LIN {X 0,Y 291.211,Z 555.04,A -85,B 0,C 180,E1 -17035.414,E2 -17035.414} C_VEL
LIN {X 0,Y 288.825,Z 546.256,A -85,B 0,C 180,E1 -17037.077,E2 -17037.077} C_VEL
LIN {X 0,Y 287.526,Z 542.188,A -85,B 0,C 180,E1 -17037.895,E2 -17037.895} C_VEL
LIN {X 0,Y 286.228,Z 538.806,A -85,B 0,C 180,E1 -17038.607,E2 -17038.607} C_VEL
LIN {X 0,Y 286.024,Z 537.383,A -85,B 0,C 180,E1 -17038.83,E2 -17038.83} C_VEL
LIN {X 0,Y 287.136,Z 533.298,A -85,B 0,C 180,E1 -17042.581,E2 -17042.581} C_VEL
LIN {X 0,Y 287.484,Z 531.734,A -85,B 0,C 180,E1 -17044.214,E2 -17044.214} C_VEL
LIN {X 0,Y 287.652,Z 529.981,A -85,B 0,C 180,E1 -17046.268,E2 -17046.268} C_VEL
LIN {X 0,Y 287.432,Z 527.724,A -85,B 0,C 180,E1 -17049.475,E2 -17049.475} C_VEL
LIN {X 0,Y 287.136,Z 525.711,A -85,B 0,C 180,E1 -17053.263,E2 -17053.263} C_VEL
LIN {X 0,Y 286.89,Z 524.296,A -85,B 0,C 180,E1 -17057.301,E2 -17057.301} C_VEL
LIN {X 0,Y 286.762,Z 523.703,A -85,B 0,C 180,E1 -17060.416,E2 -17060.416} C_VEL
LIN {X 0,Y 286.633,Z 523.532,A -85,B 0,C 180,E1 -17064.012,E2 -17064.012} C_VEL
LIN {X 0,Y 286.375,Z 523.878,A -85,B 0,C 180,E1 -17067.323,E2 -17067.323} C_VEL
LIN {X 0,Y 285.849,Z 524.654,A -85,B 0,C 180,E1 -17070.546,E2 -17070.546} C_VEL
LIN {X 0,Y 285.752,Z 524.986,A -85,B 0,C 180,E1 -17071.256,E2 -17071.256} C_VEL
LIN {X 0,Y 286.798,Z 527.778,A -85,B 0,C 180,E1 -17071.908,E2 -17071.908} C_VEL
LIN {X 0,Y 288.43,Z 530.445,A -85,B 0,C 180,E1 -17072.756,E2 -17072.756} C_VEL
LIN {X 0,Y 291.728,Z 537.483,A -85,B 0,C 180,E1 -17074.575,E2 -17074.575} C_VEL
LIN {X 0,Y 294.518,Z 545.112,A -85,B 0,C 180,E1 -17076.37,E2 -17076.37} C_VEL
LIN {X 0,Y 296.554,Z 553.072,A -85,B 0,C 180,E1 -17078.154,E2 -17078.154} C_VEL
LIN {X 0,Y 297.27,Z 559.717,A -85,B 0,C 180,E1 -17079.591,E2 -17079.591} C_VEL
LIN {X 0,Y 294.87,Z 568.726,A -85,B 0,C 180,E1 -17081.231,E2 -17081.231} C_VEL
LIN {X 0,Y 292.538,Z 575.978,A -85,B 0,C 180,E1 -17082.885,E2 -17082.885} C_VEL
LIN {X 0,Y 290.461,Z 581.891,A -85,B 0,C 180,E1 -17084.564,E2 -17084.564} C_VEL
LIN {X 0,Y 288.308,Z 587.581,A -85,B 0,C 180,E1 -17086.61,E2 -17086.61} C_VEL
LIN {X 0,Y 286.53,Z 591.939,A -85,B 0,C 180,E1 -17088.684,E2 -17088.684} C_VEL
LIN {X 0,Y 285.572,Z 594.044,A -85,B 0,C 180,E1 -17090.08,E2 -17090.08} C_VEL
LIN {X 0,Y 284.557,Z 595.665,A -85,B 0,C 180,E1 -17091.478,E2 -17091.478} C_VEL
LIN {X 0,Y 283.966,Z 596.785,A -85,B 0,C 180,E1 -17092.892,E2 -17092.892} C_VEL
LIN {X 0,Y 283.615,Z 597.465,A -85,B 0,C 180,E1 -17094.312,E2 -17094.312} C_VEL
LIN {X 0,Y 283.193,Z 597.618,A -85,B 0,C 180,E1 -17095.73,E2 -17095.73} C_VEL
LIN {X 0,Y 282.842,Z 597.22,A -85,B 0,C 180,E1 -17097.152,E2 -17097.152} C_VEL
LIN {X 0,Y 282.589,Z 596.363,A -85,B 0,C 180,E1 -17098.575,E2 -17098.575} C_VEL
LIN {X 0,Y 282.487,Z 595.035,A -85,B 0,C 180,E1 -17100,E2 -17100} C_VEL
LIN {X 0,Y 282.504,Z 591.986,A -85,B 0,C 180,E1 -17102.139,E2 -17102.139} C_VEL
LIN {X 0,Y 282.688,Z 587.669,A -85,B 0,C 180,E1 -17104.277,E2 -17104.277} C_VEL
LIN {X 0,Y 282.863,Z 582.104,A -85,B 0,C 180,E1 -17106.359,E2 -17106.359} C_VEL
LIN {X 0,Y 283.372,Z 575.719,A -85,B 0,C 180,E1 -17108.199,E2 -17108.199} C_VEL
LIN {X 0,Y 283.694,Z 569.729,A -85,B 0,C 180,E1 -17109.626,E2 -17109.626} C_VEL
LIN {X 0,Y 284.187,Z 562.583,A -85,B 0,C 180,E1 -17111.05,E2 -17111.05} C_VEL
LIN {X 0,Y 284.761,Z 555.153,A -85,B 0,C 180,E1 -17112.291,E2 -17112.291} C_VEL
LIN {X 0,Y 285.394,Z 546.206,A -85,B 0,C 180,E1 -17113.529,E2 -17113.529} C_VEL
LIN {X 0,Y 285.721,Z 538.903,A -85,B 0,C 180,E1 -17114.364,E2 -17114.364} C_VEL
LIN {X 0,Y 283.996,Z 527.158,A -85,B 0,C 180,E1 -17115.475,E2 -17115.475} C_VEL
LIN {X 0,Y 282.778,Z 517.151,A -85,B 0,C 180,E1 -17116.19,E2 -17116.19} C_VEL
LIN {X 0,Y 282.826,Z 513.933,A -85,B 0,C 180,E1 -17119.217,E2 -17119.217} C_VEL
LIN {X 0,Y 282.999,Z 510.701,A -85,B 0,C 180,E1 -17122.399,E2 -17122.399} C_VEL
LIN {X 0,Y 284.521,Z 515.556,A -85,B 0,C 180,E1 -17125.612,E2 -17125.612} C_VEL
LIN {X 0,Y 284.962,Z 519.302,A -85,B 0,C 180,E1 -17127.943,E2 -17127.943} C_VEL
LIN {X 0,Y 284.495,Z 526.168,A -85,B 0,C 180,E1 -17132.035,E2 -17132.035} C_VEL
LIN {X 0,Y 284.203,Z 530.487,A -85,B 0,C 180,E1 -17134.61,E2 -17134.61} C_VEL
LIN {X 0,Y 287.389,Z 542.62,A -85,B 0,C 180,E1 -17135.629,E2 -17135.629} C_VEL
LIN {X 0,Y 289.327,Z 553.453,A -85,B 0,C 180,E1 -17136.716,E2 -17136.716} C_VEL
LIN {X 0,Y 290.316,Z 563.05,A -85,B 0,C 180,E1 -17137.9,E2 -17137.9} C_VEL
LIN {X 0,Y 289.367,Z 571.259,A -85,B 0,C 180,E1 -17138.994,E2 -17138.994} C_VEL
LIN {X 0,Y 288.311,Z 578.189,A -85,B 0,C 180,E1 -17140.109,E2 -17140.109} C_VEL
LIN {X 0,Y 287.18,Z 584.655,A -85,B 0,C 180,E1 -17141.358,E2 -17141.358} C_VEL
LIN {X 0,Y 286.044,Z 590.927,A -85,B 0,C 180,E1 -17142.831,E2 -17142.831} C_VEL
LIN {X 0,Y 284.861,Z 597.457,A -85,B 0,C 180,E1 -17144.744,E2 -17144.744} C_VEL
LIN {X 0,Y 284.018,Z 602.375,A -85,B 0,C 180,E1 -17146.632,E2 -17146.632} C_VEL
LIN {X 0,Y 283.441,Z 605.324,A -85,B 0,C 180,E1 -17148.061,E2 -17148.061} C_VEL
LIN {X 0,Y 282.763,Z 608.747,A -85,B 0,C 180,E1 -17150.399,E2 -17150.399} C_VEL
LIN {X 0,Y 282.524,Z 609.981,A -85,B 0,C 180,E1 -17151.545,E2 -17151.545} C_VEL
LIN {X 0,Y 282.249,Z 611.122,A -85,B 0,C 180,E1 -17153.301,E2 -17153.301} C_VEL
LIN {X 0,Y 282.073,Z 611.479,A -85,B 0,C 180,E1 -17155.307,E2 -17155.307} C_VEL
LIN {X 0,Y 282.055,Z 611.13,A -85,B 0,C 180,E1 -17156.757,E2 -17156.757} C_VEL
LIN {X 0,Y 282.192,Z 610.034,A -85,B 0,C 180,E1 -17158.465,E2 -17158.465} C_VEL
LIN {X 0,Y 282.508,Z 607.716,A -85,B 0,C 180,E1 -17160.54,E2 -17160.54} C_VEL
LIN {X 0,Y 282.899,Z 604.085,A -85,B 0,C 180,E1 -17162.639,E2 -17162.639} C_VEL
LIN {X 0,Y 283.415,Z 599.288,A -85,B 0,C 180,E1 -17164.674,E2 -17164.674} C_VEL
LIN {X 0,Y 284.035,Z 594.448,A -85,B 0,C 180,E1 -17166.278,E2 -17166.278} C_VEL
LIN {X 0,Y 284.958,Z 586.826,A -85,B 0,C 180,E1 -17168.287,E2 -17168.287} C_VEL
LIN {X 0,Y 285.914,Z 578.988,A -85,B 0,C 180,E1 -17169.87,E2 -17169.87} C_VEL
LIN {X 0,Y 286.727,Z 571.873,A -85,B 0,C 180,E1 -17171.048,E2 -17171.048} C_VEL
LIN {X 0,Y 287.571,Z 563.23,A -85,B 0,C 180,E1 -17172.212,E2 -17172.212} C_VEL
LIN {X 0,Y 287.615,Z 558.748,A -85,B 0,C 180,E1 -17172.747,E2 -17172.747} C_VEL
LIN {X 0,Y 286.355,Z 548.562,A -85,B 0,C 180,E1 -17173.788,E2 -17173.788} C_VEL
LIN {X 0,Y 284.926,Z 539.502,A -85,B 0,C 180,E1 -17174.524,E2 -17174.524} C_VEL
LIN {X 0,Y 283.266,Z 530.265,A -85,B 0,C 180,E1 -17175.15,E2 -17175.15} C_VEL
LIN {X 0,Y 283.623,Z 523.602,A -85,B 0,C 180,E1 -17179.289,E2 -17179.289} C_VEL
LIN {X 0,Y 283.963,Z 516.651,A -85,B 0,C 180,E1 -17183.605,E2 -17183.605} C_VEL
LIN {X 0,Y 284.284,Z 510.406,A -85,B 0,C 180,E1 -17187.52,E2 -17187.52} C_VEL
LIN {X 0,Y 284.346,Z 509.879,A -85,B 0,C 180,E1 -17187.875,E2 -17187.875} C_VEL
LIN {X 0,Y 284.838,Z 509.818,A -85,B 0,C 180,E1 -17189.999,E2 -17189.999} C_VEL
LIN {X 0,Y 284.746,Z 509.827,A -85,B 0,C 180,E1 -17192.829,E2 -17192.829} C_VEL
LIN {X 0,Y 284.7,Z 509.832,A -85,B 0,C 180,E1 -17197.089,E2 -17197.089} C_VEL
LIN {X 0,Y 284.568,Z 509.85,A -85,B 0,C 180,E1 -17199.955,E2 -17199.955} C_VEL
LIN {X 0,Y 284.482,Z 509.863,A -85,B 0,C 180,E1 -17204.302,E2 -17204.302} C_VEL
LIN {X 0,Y 284.426,Z 509.865,A -85,B 0,C 180,E1 -17207.248,E2 -17207.248} C_VEL
LIN {X 0,Y 284.379,Z 509.876,A -85,B 0,C 180,E1 -17210.241,E2 -17210.241} C_VEL
LIN {X 0,Y 284.369,Z 509.874,A -85,B 0,C 180,E1 -17213.875,E2 -17213.875} C_VEL
LIN {X 0,Y 284.364,Z 509.877,A -85,B 0,C 180,E1 -17218.006,E2 -17218.006} C_VEL
LIN {X 0,Y 284.296,Z 509.882,A -85,B 0,C 180,E1 -17221.273,E2 -17221.273} C_VEL
LIN {X 0,Y 284.36,Z 509.873,A -85,B 0,C 180,E1 -17225.353,E2 -17225.353} C_VEL
LIN {X 0,Y 284.322,Z 509.883,A -85,B 0,C 180,E1 -17228.166,E2 -17228.166} C_VEL
LIN {X 0,Y 284.298,Z 509.884,A -85,B 0,C 180,E1 -17232.131,E2 -17232.131} C_VEL
LIN {X 0,Y 284.317,Z 509.883,A -85,B 0,C 180,E1 -17236.201,E2 -17236.201} C_VEL
LIN {X 0,Y 284.349,Z 509.879,A -85,B 0,C 180,E1 -17240.013,E2 -17240.013} C_VEL
LIN {X 0,Y 284.353,Z 509.874,A -85,B 0,C 180,E1 -17243.617,E2 -17243.617} C_VEL
LIN {X 0,Y 284.305,Z 509.88,A -85,B 0,C 180,E1 -17247.189,E2 -17247.189} C_VEL
LIN {X 0,Y 284.356,Z 509.876,A -85,B 0,C 180,E1 -17250.376,E2 -17250.376} C_VEL
LIN {X 0,Y 284.376,Z 509.873,A -85,B 0,C 180,E1 -17253.586,E2 -17253.586} C_VEL
LIN {X 0,Y 284.364,Z 509.873,A -85,B 0,C 180,E1 -17256.707,E2 -17256.707} C_VEL
LIN {X 0,Y 284.401,Z 509.868,A -85,B 0,C 180,E1 -17261.261,E2 -17261.261} C_VEL
LIN {X 0,Y 284.49,Z 509.858,A -85,B 0,C 180,E1 -17264.459,E2 -17264.459} C_VEL
LIN {X 0,Y 284.487,Z 509.857,A -85,B 0,C 180,E1 -17268.601,E2 -17268.601} C_VEL
LIN {X 0,Y 284.657,Z 509.839,A -85,B 0,C 180,E1 -17271.481,E2 -17271.481} C_VEL
LIN {X 0,Y 284.6,Z 509.845,A -85,B 0,C 180,E1 -17274.331,E2 -17274.331} C_VEL
LIN {X 0,Y 284.855,Z 509.809,A -85,B 0,C 180,E1 -17278.586,E2 -17278.586} C_VEL
LIN {X 0,Y 284.854,Z 509.813,A -85,B 0,C 180,E1 -17281.414,E2 -17281.414} C_VEL
LIN {X 0,Y 284.522,Z 509.854,A -85,B 0,C 180,E1 -17284.135,E2 -17284.135} C_VEL
LIN {X 0,Y 283.792,Z 509.952,A -85,B 0,C 180,E1 -17285.317,E2 -17285.317} C_VEL
LIN {X 0,Y 280.998,Z 510.303,A -85,B 0,C 180,E1 -17287.245,E2 -17287.245} C_VEL
LIN {X 0,Y 277.838,Z 510.69,A -85,B 0,C 180,E1 -17289.614,E2 -17289.614} C_VEL
LIN {X 0,Y 277.482,Z 510.731,A -85,B 0,C 180,E1 -17290.431,E2 -17290.431} C_VEL
LIN {X 0,Y 277.432,Z 510.737,A -85,B 0,C 180,E1 -17294.674,E2 -17294.674} C_VEL
LIN {X 0,Y 277.342,Z 510.75,A -85,B 0,C 180,E1 -17299.234,E2 -17299.234} C_VEL
LIN {X 0,Y 277.326,Z 510.753,A -85,B 0,C 180,E1 -17303.921,E2 -17303.921} C_VEL
LIN {X 0,Y 277.323,Z 510.755,A -85,B 0,C 180,E1 -17307.506,E2 -17307.506} C_VEL
LIN {X 0,Y 277.269,Z 510.758,A -85,B 0,C 180,E1 -17310.482,E2 -17310.482} C_VEL
LIN {X 0,Y 277.252,Z 510.761,A -85,B 0,C 180,E1 -17313.895,E2 -17313.895} C_VEL
LIN {X 0,Y 277.279,Z 510.76,A -85,B 0,C 180,E1 -17317.467,E2 -17317.467} C_VEL
LIN {X 0,Y 277.224,Z 510.766,A -85,B 0,C 180,E1 -17321.234,E2 -17321.234} C_VEL
LIN {X 0,Y 277.231,Z 510.765,A -85,B 0,C 180,E1 -17325.22,E2 -17325.22} C_VEL
LIN {X 0,Y 277.285,Z 510.76,A -85,B 0,C 180,E1 -17329.497,E2 -17329.497} C_VEL
LIN {X 0,Y 277.513,Z 510.799,A -85,B 0,C 180,E1 -17332.163,E2 -17332.163} C_VEL
LIN {X 0,Y 278.528,Z 516.826,A -85,B 0,C 180,E1 -17336.375,E2 -17336.375} C_VEL
LIN {X 0,Y 278.767,Z 519.283,A -85,B 0,C 180,E1 -17338.034,E2 -17338.034} C_VEL
LIN {X 0,Y 277.963,Z 524.259,A -85,B 0,C 180,E1 -17341.29,E2 -17341.29} C_VEL
LIN {X 0,Y 276.905,Z 531.592,A -85,B 0,C 180,E1 -17346.042,E2 -17346.042} C_VEL
LIN {X 0,Y 276.175,Z 538.547,A -85,B 0,C 180,E1 -17350.515,E2 -17350.515} C_VEL
LIN {X 0,Y 277.843,Z 552.725,A -85,B 0,C 180,E1 -17351.234,E2 -17351.234} C_VEL
LIN {X 0,Y 278.722,Z 562.025,A -85,B 0,C 180,E1 -17351.914,E2 -17351.914} C_VEL
LIN {X 0,Y 279.238,Z 570.27,A -85,B 0,C 180,E1 -17352.681,E2 -17352.681} C_VEL
LIN {X 0,Y 279.551,Z 579.34,A -85,B 0,C 180,E1 -17353.732,E2 -17353.732} C_VEL
LIN {X 0,Y 279.2,Z 586.143,A -85,B 0,C 180,E1 -17354.675,E2 -17354.675} C_VEL
LIN {X 0,Y 278.266,Z 593.763,A -85,B 0,C 180,E1 -17355.932,E2 -17355.932} C_VEL
LIN {X 0,Y 277.355,Z 601.745,A -85,B 0,C 180,E1 -17357.563,E2 -17357.563} C_VEL
LIN {X 0,Y 276.494,Z 608.666,A -85,B 0,C 180,E1 -17359.381,E2 -17359.381} C_VEL
LIN {X 0,Y 275.949,Z 614.155,A -85,B 0,C 180,E1 -17361.211,E2 -17361.211} C_VEL
LIN {X 0,Y 275.503,Z 619.232,A -85,B 0,C 180,E1 -17363.409,E2 -17363.409} C_VEL
LIN {X 0,Y 275.325,Z 622.886,A -85,B 0,C 180,E1 -17365.609,E2 -17365.609} C_VEL
LIN {X 0,Y 275.323,Z 624.523,A -85,B 0,C 180,E1 -17367.074,E2 -17367.074} C_VEL
LIN {X 0,Y 275.3,Z 625.615,A -85,B 0,C 180,E1 -17368.538,E2 -17368.538} C_VEL
LIN {X 0,Y 275.325,Z 626.211,A -85,B 0,C 180,E1 -17370.001,E2 -17370.001} C_VEL
LIN {X 0,Y 275.297,Z 626.32,A -85,B 0,C 180,E1 -17371.464,E2 -17371.464} C_VEL
LIN {X 0,Y 275.314,Z 625.931,A -85,B 0,C 180,E1 -17372.927,E2 -17372.927} C_VEL
LIN {X 0,Y 275.319,Z 624.951,A -85,B 0,C 180,E1 -17374.393,E2 -17374.393} C_VEL
LIN {X 0,Y 275.524,Z 622.567,A -85,B 0,C 180,E1 -17376.592,E2 -17376.592} C_VEL
LIN {X 0,Y 275.695,Z 621.412,A -85,B 0,C 180,E1 -17377.324,E2 -17377.324} C_VEL
LIN {X 0,Y 276.68,Z 617.967,A -85,B 0,C 180,E1 -17380.243,E2 -17380.243} C_VEL
LIN {X 0,Y 277.921,Z 614.293,A -85,B 0,C 180,E1 -17382.413,E2 -17382.413} C_VEL
LIN {X 0,Y 279.712,Z 609.31,A -85,B 0,C 180,E1 -17384.553,E2 -17384.553} C_VEL
LIN {X 0,Y 281.526,Z 604.159,A -85,B 0,C 180,E1 -17386.311,E2 -17386.311} C_VEL
LIN {X 0,Y 283.064,Z 599.285,A -85,B 0,C 180,E1 -17387.708,E2 -17387.708} C_VEL
LIN {X 0,Y 285.508,Z 591.962,A -85,B 0,C 180,E1 -17389.41,E2 -17389.41} C_VEL
LIN {X 0,Y 287.159,Z 584.573,A -85,B 0,C 180,E1 -17390.942,E2 -17390.942} C_VEL
LIN {X 0,Y 287.682,Z 577.918,A -85,B 0,C 180,E1 -17392.251,E2 -17392.251} C_VEL
LIN {X 0,Y 287.227,Z 567.044,A -85,B 0,C 180,E1 -17394.369,E2 -17394.369} C_VEL
LIN {X 0,Y 285.224,Z 555.475,A -85,B 0,C 180,E1 -17396.633,E2 -17396.633} C_VEL
LIN {X 0,Y 283.08,Z 547.236,A -85,B 0,C 180,E1 -17398.356,E2 -17398.356} C_VEL
LIN {X 0,Y 281.383,Z 541.883,A -85,B 0,C 180,E1 -17399.585,E2 -17399.585} C_VEL
LIN {X 0,Y 279.978,Z 538.608,A -85,B 0,C 180,E1 -17400.431,E2 -17400.431} C_VEL
LIN {X 0,Y 279.641,Z 536.505,A -85,B 0,C 180,E1 -17400.87,E2 -17400.87} C_VEL
LIN {X 0,Y 280.553,Z 533.19,A -85,B 0,C 180,E1 -17404.242,E2 -17404.242} C_VEL
LIN {X 0,Y 280.668,Z 531.012,A -85,B 0,C 180,E1 -17406.94,E2 -17406.94} C_VEL
LIN {X 0,Y 280.419,Z 528.637,A -85,B 0,C 180,E1 -17410.665,E2 -17410.665} C_VEL
LIN {X 0,Y 280.162,Z 526.796,A -85,B 0,C 180,E1 -17414.62,E2 -17414.62} C_VEL
LIN {X 0,Y 279.985,Z 525.939,A -85,B 0,C 180,E1 -17417.333,E2 -17417.333} C_VEL
LIN {X 0,Y 279.822,Z 525.264,A -85,B 0,C 180,E1 -17421.133,E2 -17421.133} C_VEL
LIN {X 0,Y 279.635,Z 525.177,A -85,B 0,C 180,E1 -17424.686,E2 -17424.686} C_VEL
LIN {X 0,Y 279.316,Z 525.596,A -85,B 0,C 180,E1 -17428.103,E2 -17428.103} C_VEL
LIN {X 0,Y 279.229,Z 525.917,A -85,B 0,C 180,E1 -17429.208,E2 -17429.208} C_VEL
LIN {X 0,Y 280.088,Z 528.435,A -85,B 0,C 180,E1 -17429.878,E2 -17429.878} C_VEL
LIN {X 0,Y 281.728,Z 530.717,A -85,B 0,C 180,E1 -17430.824,E2 -17430.824} C_VEL
LIN {X 0,Y 285.489,Z 538.633,A -85,B 0,C 180,E1 -17433.195,E2 -17433.195} C_VEL
LIN {X 0,Y 288.139,Z 545.714,A -85,B 0,C 180,E1 -17435.074,E2 -17435.074} C_VEL
LIN {X 0,Y 290.208,Z 553.385,A -85,B 0,C 180,E1 -17436.964,E2 -17436.964} C_VEL
LIN {X 0,Y 291.107,Z 559.638,A -85,B 0,C 180,E1 -17438.451,E2 -17438.451} C_VEL
LIN {X 0,Y 291.107,Z 562.823,A -85,B 0,C 180,E1 -17439.139,E2 -17439.139} C_VEL
LIN {X 0,Y 288.431,Z 571.16,A -85,B 0,C 180,E1 -17440.795,E2 -17440.795} C_VEL
LIN {X 0,Y 286.006,Z 577.979,A -85,B 0,C 180,E1 -17442.481,E2 -17442.481} C_VEL
LIN {X 0,Y 283.824,Z 583.652,A -85,B 0,C 180,E1 -17444.194,E2 -17444.194} C_VEL
LIN {X 0,Y 281.553,Z 589.068,A -85,B 0,C 180,E1 -17446.283,E2 -17446.283} C_VEL
LIN {X 0,Y 279.655,Z 593.016,A -85,B 0,C 180,E1 -17448.402,E2 -17448.402} C_VEL
LIN {X 0,Y 278.651,Z 595.054,A -85,B 0,C 180,E1 -17449.831,E2 -17449.831} C_VEL
LIN {X 0,Y 277.602,Z 596.516,A -85,B 0,C 180,E1 -17451.263,E2 -17451.263} C_VEL
LIN {X 0,Y 276.958,Z 597.456,A -85,B 0,C 180,E1 -17452.711,E2 -17452.711} C_VEL
LIN {X 0,Y 276.566,Z 597.945,A -85,B 0,C 180,E1 -17454.166,E2 -17454.166} C_VEL
LIN {X 0,Y 276.131,Z 598.009,A -85,B 0,C 180,E1 -17455.621,E2 -17455.621} C_VEL
LIN {X 0,Y 275.768,Z 597.514,A -85,B 0,C 180,E1 -17457.078,E2 -17457.078} C_VEL
LIN {X 0,Y 275.508,Z 596.486,A -85,B 0,C 180,E1 -17458.538,E2 -17458.538} C_VEL
LIN {X 0,Y 275.404,Z 594.989,A -85,B 0,C 180,E1 -17460,E2 -17460} C_VEL
LIN {X 0,Y 275.431,Z 591.762,A -85,B 0,C 180,E1 -17462.194,E2 -17462.194} C_VEL
LIN {X 0,Y 275.609,Z 587.285,A -85,B 0,C 180,E1 -17464.388,E2 -17464.388} C_VEL
LIN {X 0,Y 275.776,Z 582.036,A -85,B 0,C 180,E1 -17466.33,E2 -17466.33} C_VEL
LIN {X 0,Y 276.255,Z 576.21,A -85,B 0,C 180,E1 -17468.043,E2 -17468.043} C_VEL
LIN {X 0,Y 276.545,Z 570.229,A -85,B 0,C 180,E1 -17469.508,E2 -17469.508} C_VEL
LIN {X 0,Y 277.073,Z 563.111,A -85,B 0,C 180,E1 -17470.967,E2 -17470.967} C_VEL
LIN {X 0,Y 277.715,Z 554.54,A -85,B 0,C 180,E1 -17472.422,E2 -17472.422} C_VEL
LIN {X 0,Y 278.479,Z 544.006,A -85,B 0,C 180,E1 -17473.872,E2 -17473.872} C_VEL
LIN {X 0,Y 278.594,Z 539.019,A -85,B 0,C 180,E1 -17474.425,E2 -17474.425} C_VEL
LIN {X 0,Y 276.917,Z 527.605,A -85,B 0,C 180,E1 -17475.534,E2 -17475.534} C_VEL
LIN {X 0,Y 275.698,Z 517.493,A -85,B 0,C 180,E1 -17476.285,E2 -17476.285} C_VEL
LIN {X 0,Y 275.741,Z 514.209,A -85,B 0,C 180,E1 -17479.428,E2 -17479.428} C_VEL
LIN {X 0,Y 275.868,Z 511.733,A -85,B 0,C 180,E1 -17481.924,E2 -17481.924} C_VEL
LIN {X 0,Y 277.571,Z 516.984,A -85,B 0,C 180,E1 -17485.495,E2 -17485.495} C_VEL
LIN {X 0,Y 278.021,Z 520.527,A -85,B 0,C 180,E1 -17487.777,E2 -17487.777} C_VEL
LIN {X 0,Y 277.505,Z 527.693,A -85,B 0,C 180,E1 -17492.13,E2 -17492.13} C_VEL
LIN {X 0,Y 277.289,Z 530.831,A -85,B 0,C 180,E1 -17493.945,E2 -17493.945} C_VEL
LIN {X 0,Y 280.094,Z 540.854,A -85,B 0,C 180,E1 -17494.808,E2 -17494.808} C_VEL
LIN {X 0,Y 281.952,Z 549.804,A -85,B 0,C 180,E1 -17495.712,E2 -17495.712} C_VEL
LIN {X 0,Y 283.431,Z 560.979,A -85,B 0,C 180,E1 -17497.033,E2 -17497.033} C_VEL
LIN {X 0,Y 283.585,Z 565.7,A -85,B 0,C 180,E1 -17497.685,E2 -17497.685} C_VEL
LIN {X 0,Y 282.101,Z 575.692,A -85,B 0,C 180,E1 -17499.136,E2 -17499.136} C_VEL
LIN {X 0,Y 280.706,Z 583.539,A -85,B 0,C 180,E1 -17500.614,E2 -17500.614} C_VEL
LIN {X 0,Y 279.484,Z 589.911,A -85,B 0,C 180,E1 -17502.087,E2 -17502.087} C_VEL
LIN {X 0,Y 278.529,Z 594.928,A -85,B 0,C 180,E1 -17503.494,E2 -17503.494} C_VEL
LIN {X 0,Y 277.593,Z 599.734,A -85,B 0,C 180,E1 -17505.145,E2 -17505.145} C_VEL
LIN {X 0,Y 276.862,Z 603.456,A -85,B 0,C 180,E1 -17506.734,E2 -17506.734} C_VEL
LIN {X 0,Y 276.198,Z 606.799,A -85,B 0,C 180,E1 -17508.578,E2 -17508.578} C_VEL
LIN {X 0,Y 275.685,Z 609.201,A -85,B 0,C 180,E1 -17510.407,E2 -17510.407} C_VEL
LIN {X 0,Y 275.32,Z 610.81,A -85,B 0,C 180,E1 -17512.31,E2 -17512.31} C_VEL
LIN {X 0,Y 275.005,Z 611.686,A -85,B 0,C 180,E1 -17514.864,E2 -17514.864} C_VEL
LIN {X 0,Y 275.012,Z 610.826,A -85,B 0,C 180,E1 -17517.543,E2 -17517.543} C_VEL
LIN {X 0,Y 275.374,Z 608.378,A -85,B 0,C 180,E1 -17520.197,E2 -17520.197} C_VEL
LIN {X 0,Y 275.83,Z 604.317,A -85,B 0,C 180,E1 -17522.7,E2 -17522.7} C_VEL
LIN {X 0,Y 276.214,Z 600.612,A -85,B 0,C 180,E1 -17524.37,E2 -17524.37} C_VEL
LIN {X 0,Y 276.846,Z 595.913,A -85,B 0,C 180,E1 -17526.05,E2 -17526.05} C_VEL
LIN {X 0,Y 277.541,Z 590.292,A -85,B 0,C 180,E1 -17527.676,E2 -17527.676} C_VEL
LIN {X 0,Y 278.312,Z 584.201,A -85,B 0,C 180,E1 -17529.121,E2 -17529.121} C_VEL
LIN {X 0,Y 279.177,Z 577.064,A -85,B 0,C 180,E1 -17530.515,E2 -17530.515} C_VEL
LIN {X 0,Y 280.286,Z 567.591,A -85,B 0,C 180,E1 -17532.003,E2 -17532.003} C_VEL
LIN {X 0,Y 280.754,Z 560.552,A -85,B 0,C 180,E1 -17532.894,E2 -17532.894} C_VEL
LIN {X 0,Y 279.468,Z 549.59,A -85,B 0,C 180,E1 -17534.076,E2 -17534.076} C_VEL
LIN {X 0,Y 277.943,Z 539.973,A -85,B 0,C 180,E1 -17534.892,E2 -17534.892} C_VEL
LIN {X 0,Y 276.226,Z 530.431,A -85,B 0,C 180,E1 -17535.533,E2 -17535.533} C_VEL
LIN {X 0,Y 276.614,Z 523.757,A -85,B 0,C 180,E1 -17539.755,E2 -17539.755} C_VEL
LIN {X 0,Y 276.913,Z 517.912,A -85,B 0,C 180,E1 -17543.441,E2 -17543.441} C_VEL
LIN {X 0,Y 277.195,Z 512.161,A -85,B 0,C 180,E1 -17547.093,E2 -17547.093} C_VEL
LIN {X 0,Y 277.335,Z 510.753,A -85,B 0,C 180,E1 -17548.002,E2 -17548.002} C_VEL
LIN {X 0,Y 277.796,Z 510.695,A -85,B 0,C 180,E1 -17549.999,E2 -17549.999} C_VEL
LIN {X 0,Y 277.702,Z 510.705,A -85,B 0,C 180,E1 -17552.901,E2 -17552.901} C_VEL
LIN {X 0,Y 277.655,Z 510.709,A -85,B 0,C 180,E1 -17557.27,E2 -17557.27} C_VEL
LIN {X 0,Y 277.508,Z 510.732,A -85,B 0,C 180,E1 -17560.21,E2 -17560.21} C_VEL
LIN {X 0,Y 277.435,Z 510.738,A -85,B 0,C 180,E1 -17564.673,E2 -17564.673} C_VEL
LIN {X 0,Y 277.345,Z 510.747,A -85,B 0,C 180,E1 -17569.233,E2 -17569.233} C_VEL
LIN {X 0,Y 277.319,Z 510.754,A -85,B 0,C 180,E1 -17574.17,E2 -17574.17} C_VEL
LIN {X 0,Y 277.335,Z 510.749,A -85,B 0,C 180,E1 -17577.508,E2 -17577.508} C_VEL
LIN {X 0,Y 277.271,Z 510.759,A -85,B 0,C 180,E1 -17580.481,E2 -17580.481} C_VEL
LIN {X 0,Y 277.253,Z 510.761,A -85,B 0,C 180,E1 -17583.894,E2 -17583.894} C_VEL
LIN {X 0,Y 277.28,Z 510.756,A -85,B 0,C 180,E1 -17587.466,E2 -17587.466} C_VEL
LIN {X 0,Y 277.233,Z 510.761,A -85,B 0,C 180,E1 -17591.231,E2 -17591.231} C_VEL
LIN {X 0,Y 277.249,Z 510.759,A -85,B 0,C 180,E1 -17595.215,E2 -17595.215} C_VEL
LIN {X 0,Y 277.293,Z 510.755,A -85,B 0,C 180,E1 -17599.494,E2 -17599.494} C_VEL
LIN {X 0,Y 277.288,Z 510.753,A -85,B 0,C 180,E1 -17602.534,E2 -17602.534} C_VEL
LIN {X 0,Y 277.252,Z 510.763,A -85,B 0,C 180,E1 -17606.105,E2 -17606.105} C_VEL
LIN {X 0,Y 277.259,Z 510.76,A -85,B 0,C 180,E1 -17609.538,E2 -17609.538} C_VEL
LIN {X 0,Y 277.356,Z 510.745,A -85,B 0,C 180,E1 -17612.864,E2 -17612.864} C_VEL
LIN {X 0,Y 277.326,Z 510.754,A -85,B 0,C 180,E1 -17616.079,E2 -17616.079} C_VEL
LIN {X 0,Y 277.342,Z 510.746,A -85,B 0,C 180,E1 -17620.766,E2 -17620.766} C_VEL
LIN {X 0,Y 277.432,Z 510.738,A -85,B 0,C 180,E1 -17625.326,E2 -17625.326} C_VEL
LIN {X 0,Y 277.505,Z 510.731,A -85,B 0,C 180,E1 -17629.789,E2 -17629.789} C_VEL
LIN {X 0,Y 277.651,Z 510.709,A -85,B 0,C 180,E1 -17632.729,E2 -17632.729} C_VEL
LIN {X 0,Y 277.821,Z 510.685,A -85,B 0,C 180,E1 -17638.55,E2 -17638.55} C_VEL
LIN {X 0,Y 277.819,Z 510.689,A -85,B 0,C 180,E1 -17641.449,E2 -17641.449} C_VEL
LIN {X 0,Y 277.651,Z 510.71,A -85,B 0,C 180,E1 -17647.271,E2 -17647.271} C_VEL
LIN {X 0,Y 277.482,Z 510.731,A -85,B 0,C 180,E1 -17650.431,E2 -17650.431} C_VEL
LIN {X 0,Y 276.754,Z 510.826,A -85,B 0,C 180,E1 -17651.641,E2 -17651.641} C_VEL
LIN {X 0,Y 273.911,Z 511.18,A -85,B 0,C 180,E1 -17653.614,E2 -17653.614} C_VEL
LIN {X 0,Y 271.509,Z 511.478,A -85,B 0,C 180,E1 -17655.216,E2 -17655.216} C_VEL
LIN {X 0,Y 270.438,Z 511.608,A -85,B 0,C 180,E1 -17656.457,E2 -17656.457} C_VEL
LIN {X 0,Y 270.327,Z 511.62,A -85,B 0,C 180,E1 -17656.878,E2 -17656.878} C_VEL
LIN {X 0,Y 270.29,Z 511.627,A -85,B 0,C 180,E1 -17660.602,E2 -17660.602} C_VEL
LIN {X 0,Y 270.271,Z 511.629,A -85,B 0,C 180,E1 -17664.586,E2 -17664.586} C_VEL
LIN {X 0,Y 270.267,Z 511.632,A -85,B 0,C 180,E1 -17667.909,E2 -17667.909} C_VEL
LIN {X 0,Y 270.182,Z 511.643,A -85,B 0,C 180,E1 -17671.348,E2 -17671.348} C_VEL
LIN {X 0,Y 270.212,Z 511.637,A -85,B 0,C 180,E1 -17674.904,E2 -17674.904} C_VEL
LIN {X 0,Y 270.219,Z 511.635,A -85,B 0,C 180,E1 -17678.717,E2 -17678.717} C_VEL
LIN {X 0,Y 270.189,Z 511.64,A -85,B 0,C 180,E1 -17682.555,E2 -17682.555} C_VEL
LIN {X 0,Y 270.195,Z 511.639,A -85,B 0,C 180,E1 -17686.744,E2 -17686.744} C_VEL
LIN {X 0,Y 270.426,Z 511.613,A -85,B 0,C 180,E1 -17691.887,E2 -17691.887} C_VEL
LIN {X 0,Y 270.496,Z 511.898,A -85,B 0,C 180,E1 -17692.37,E2 -17692.37} C_VEL
LIN {X 0,Y 271.355,Z 516.902,A -85,B 0,C 180,E1 -17695.974,E2 -17695.974} C_VEL
LIN {X 0,Y 271.684,Z 519.735,A -85,B 0,C 180,E1 -17697.956,E2 -17697.956} C_VEL
LIN {X 0,Y 270.853,Z 524.703,A -85,B 0,C 180,E1 -17701.3,E2 -17701.3} C_VEL
LIN {X 0,Y 269.858,Z 531.321,A -85,B 0,C 180,E1 -17705.716,E2 -17705.716} C_VEL
LIN {X 0,Y 269.118,Z 537.883,A -85,B 0,C 180,E1 -17710.074,E2 -17710.074} C_VEL
LIN {X 0,Y 270.83,Z 552.126,A -85,B 0,C 180,E1 -17710.803,E2 -17710.803} C_VEL
LIN {X 0,Y 271.71,Z 561.831,A -85,B 0,C 180,E1 -17711.528,E2 -17711.528} C_VEL
LIN {X 0,Y 272.284,Z 570.584,A -85,B 0,C 180,E1 -17712.373,E2 -17712.373} C_VEL
LIN {X 0,Y 272.543,Z 578.73,A -85,B 0,C 180,E1 -17713.344,E2 -17713.344} C_VEL
LIN {X 0,Y 272.446,Z 584.136,A -85,B 0,C 180,E1 -17714.094,E2 -17714.094} C_VEL
LIN {X 0,Y 271.515,Z 592.063,A -85,B 0,C 180,E1 -17715.383,E2 -17715.383} C_VEL
LIN {X 0,Y 270.783,Z 597.757,A -85,B 0,C 180,E1 -17716.492,E2 -17716.492} C_VEL
LIN {X 0,Y 270.025,Z 604.102,A -85,B 0,C 180,E1 -17717.983,E2 -17717.983} C_VEL
LIN {X 0,Y 269.356,Z 609.357,A -85,B 0,C 180,E1 -17719.477,E2 -17719.477} C_VEL
LIN {X 0,Y 268.91,Z 613.727,A -85,B 0,C 180,E1 -17720.979,E2 -17720.979} C_VEL
LIN {X 0,Y 268.425,Z 618.852,A -85,B 0,C 180,E1 -17723.234,E2 -17723.234} C_VEL
LIN {X 0,Y 268.236,Z 622.569,A -85,B 0,C 180,E1 -17725.493,E2 -17725.493} C_VEL
LIN {X 0,Y 268.233,Z 624.232,A -85,B 0,C 180,E1 -17726.997,E2 -17726.997} C_VEL
LIN {X 0,Y 268.226,Z 625.365,A -85,B 0,C 180,E1 -17728.499,E2 -17728.499} C_VEL
LIN {X 0,Y 268.247,Z 626,A -85,B 0,C 180,E1 -17730.001,E2 -17730.001} C_VEL
LIN {X 0,Y 268.223,Z 626.148,A -85,B 0,C 180,E1 -17731.502,E2 -17731.502} C_VEL
LIN {X 0,Y 268.225,Z 625.777,A -85,B 0,C 180,E1 -17733.005,E2 -17733.005} C_VEL
LIN {X 0,Y 268.344,Z 623.805,A -85,B 0,C 180,E1 -17735.6,E2 -17735.6} C_VEL
LIN {X 0,Y 270.111,Z 617.084,A -85,B 0,C 180,E1 -17741.254,E2 -17741.254} C_VEL
LIN {X 0,Y 271.567,Z 613.248,A -85,B 0,C 180,E1 -17743.47,E2 -17743.47} C_VEL
LIN {X 0,Y 273.593,Z 608.153,A -85,B 0,C 180,E1 -17745.648,E2 -17745.648} C_VEL
LIN {X 0,Y 275.975,Z 601.737,A -85,B 0,C 180,E1 -17747.795,E2 -17747.795} C_VEL
LIN {X 0,Y 279.009,Z 593.684,A -85,B 0,C 180,E1 -17749.881,E2 -17749.881} C_VEL
LIN {X 0,Y 280.934,Z 585.76,A -85,B 0,C 180,E1 -17751.621,E2 -17751.621} C_VEL
LIN {X 0,Y 281.616,Z 578.613,A -85,B 0,C 180,E1 -17753.145,E2 -17753.145} C_VEL
LIN {X 0,Y 281.449,Z 570.414,A -85,B 0,C 180,E1 -17754.845,E2 -17754.845} C_VEL
LIN {X 0,Y 280.552,Z 562.568,A -85,B 0,C 180,E1 -17756.518,E2 -17756.518} C_VEL
LIN {X 0,Y 278.525,Z 552.333,A -85,B 0,C 180,E1 -17758.797,E2 -17758.797} C_VEL
LIN {X 0,Y 276.764,Z 546.257,A -85,B 0,C 180,E1 -17760.302,E2 -17760.302} C_VEL
LIN {X 0,Y 275.374,Z 541.493,A -85,B 0,C 180,E1 -17761.548,E2 -17761.548} C_VEL
LIN {X 0,Y 273.874,Z 538.276,A -85,B 0,C 180,E1 -17762.609,E2 -17762.609} C_VEL
LIN {X 0,Y 273.371,Z 535.513,A -85,B 0,C 180,E1 -17763.335,E2 -17763.335} C_VEL
LIN {X 0,Y 273.642,Z 534.282,A -85,B 0,C 180,E1 -17764.729,E2 -17764.729} C_VEL
LIN {X 0,Y 273.662,Z 531.82,A -85,B 0,C 180,E1 -17768.051,E2 -17768.051} C_VEL
LIN {X 0,Y 273.392,Z 529.601,A -85,B 0,C 180,E1 -17771.943,E2 -17771.943} C_VEL
LIN {X 0,Y 273.301,Z 528.69,A -85,B 0,C 180,E1 -17773.973,E2 -17773.973} C_VEL
LIN {X 0,Y 273.016,Z 527.435,A -85,B 0,C 180,E1 -17777.988,E2 -17777.988} C_VEL
LIN {X 0,Y 272.864,Z 526.851,A -85,B 0,C 180,E1 -17781.819,E2 -17781.819} C_VEL
LIN {X 0,Y 272.661,Z 526.836,A -85,B 0,C 180,E1 -17785.455,E2 -17785.455} C_VEL
LIN {X 0,Y 272.586,Z 527.02,A -85,B 0,C 180,E1 -17786.601,E2 -17786.601} C_VEL
LIN {X 0,Y 273.317,Z 529.167,A -85,B 0,C 180,E1 -17787.317,E2 -17787.317} C_VEL
LIN {X 0,Y 275.56,Z 532.088,A -85,B 0,C 180,E1 -17788.862,E2 -17788.862} C_VEL
LIN {X 0,Y 276.648,Z 534.722,A -85,B 0,C 180,E1 -17789.74,E2 -17789.74} C_VEL
LIN {X 0,Y 277.822,Z 536.506,A -85,B 0,C 180,E1 -17790.473,E2 -17790.473} C_VEL
LIN {X 0,Y 281.177,Z 544.704,A -85,B 0,C 180,E1 -17793.084,E2 -17793.084} C_VEL
LIN {X 0,Y 283.432,Z 551.656,A -85,B 0,C 180,E1 -17795.069,E2 -17795.069} C_VEL
LIN {X 0,Y 284.913,Z 559.258,A -85,B 0,C 180,E1 -17797.086,E2 -17797.086} C_VEL
LIN {X 0,Y 285.219,Z 564.12,A -85,B 0,C 180,E1 -17798.308,E2 -17798.308} C_VEL
LIN {X 0,Y 283.695,Z 569.101,A -85,B 0,C 180,E1 -17799.328,E2 -17799.328} C_VEL
LIN {X 0,Y 281.012,Z 576.419,A -85,B 0,C 180,E1 -17801.027,E2 -17801.027} C_VEL
LIN {X 0,Y 278.519,Z 582.358,A -85,B 0,C 180,E1 -17802.753,E2 -17802.753} C_VEL
LIN {X 0,Y 276.348,Z 587.183,A -85,B 0,C 180,E1 -17804.512,E2 -17804.512} C_VEL
LIN {X 0,Y 274.089,Z 591.786,A -85,B 0,C 180,E1 -17806.658,E2 -17806.658} C_VEL
LIN {X 0,Y 272.559,Z 594.634,A -85,B 0,C 180,E1 -17808.478,E2 -17808.478} C_VEL
LIN {X 0,Y 270.635,Z 597.34,A -85,B 0,C 180,E1 -17811.036,E2 -17811.036} C_VEL
LIN {X 0,Y 269.956,Z 598.123,A -85,B 0,C 180,E1 -17812.521,E2 -17812.521} C_VEL
LIN {X 0,Y 269.522,Z 598.429,A -85,B 0,C 180,E1 -17814.013,E2 -17814.013} C_VEL
LIN {X 0,Y 269.073,Z 598.307,A -85,B 0,C 180,E1 -17815.506,E2 -17815.506} C_VEL
LIN {X 0,Y 268.696,Z 597.735,A -85,B 0,C 180,E1 -17817.002,E2 -17817.002} C_VEL
LIN {X 0,Y 268.429,Z 596.598,A -85,B 0,C 180,E1 -17818.5,E2 -17818.5} C_VEL
LIN {X 0,Y 268.298,Z 593.984,A -85,B 0,C 180,E1 -17820.751,E2 -17820.751} C_VEL
LIN {X 0,Y 268.444,Z 590.05,A -85,B 0,C 180,E1 -17823.002,E2 -17823.002} C_VEL
LIN {X 0,Y 268.534,Z 585.289,A -85,B 0,C 180,E1 -17825.053,E2 -17825.053} C_VEL
LIN {X 0,Y 268.748,Z 580.598,A -85,B 0,C 180,E1 -17826.683,E2 -17826.683} C_VEL
LIN {X 0,Y 269.209,Z 575.172,A -85,B 0,C 180,E1 -17828.255,E2 -17828.255} C_VEL
LIN {X 0,Y 269.544,Z 568.99,A -85,B 0,C 180,E1 -17829.758,E2 -17829.758} C_VEL
LIN {X 0,Y 270.063,Z 561.645,A -85,B 0,C 180,E1 -17831.255,E2 -17831.255} C_VEL
LIN {X 0,Y 270.9,Z 551.526,A -85,B 0,C 180,E1 -17832.93,E2 -17832.93} C_VEL
LIN {X 0,Y 271.546,Z 541.384,A -85,B 0,C 180,E1 -17834.234,E2 -17834.234} C_VEL
LIN {X 0,Y 270.618,Z 533.79,A -85,B 0,C 180,E1 -17835.053,E2 -17835.053} C_VEL
LIN {X 0,Y 269.314,Z 524.184,A -85,B 0,C 180,E1 -17835.898,E2 -17835.898} C_VEL
LIN {X 0,Y 268.62,Z 517.826,A -85,B 0,C 180,E1 -17836.377,E2 -17836.377} C_VEL
LIN {X 0,Y 268.708,Z 513.028,A -85,B 0,C 180,E1 -17841.078,E2 -17841.078} C_VEL
LIN {X 0,Y 268.748,Z 512.867,A -85,B 0,C 180,E1 -17841.476,E2 -17841.476} C_VEL
LIN {X 0,Y 270.611,Z 518.428,A -85,B 0,C 180,E1 -17845.374,E2 -17845.374} C_VEL
LIN {X 0,Y 271.059,Z 520.845,A -85,B 0,C 180,E1 -17846.984,E2 -17846.984} C_VEL
LIN {X 0,Y 270.722,Z 526.125,A -85,B 0,C 180,E1 -17850.281,E2 -17850.281} C_VEL
LIN {X 0,Y 270.392,Z 530.822,A -85,B 0,C 180,E1 -17853.194,E2 -17853.194} C_VEL
LIN {X 0,Y 273.287,Z 541.073,A -85,B 0,C 180,E1 -17854.123,E2 -17854.123} C_VEL
LIN {X 0,Y 275.32,Z 550.745,A -85,B 0,C 180,E1 -17855.144,E2 -17855.144} C_VEL
LIN {X 0,Y 276.697,Z 561.067,A -85,B 0,C 180,E1 -17856.421,E2 -17856.421} C_VEL
LIN {X 0,Y 276.934,Z 566.48,A -85,B 0,C 180,E1 -17857.2,E2 -17857.2} C_VEL
LIN {X 0,Y 275.453,Z 575.891,A -85,B 0,C 180,E1 -17858.612,E2 -17858.612} C_VEL
LIN {X 0,Y 273.87,Z 584.373,A -85,B 0,C 180,E1 -17860.266,E2 -17860.266} C_VEL
LIN {X 0,Y 272.713,Z 590.13,A -85,B 0,C 180,E1 -17861.638,E2 -17861.638} C_VEL
LIN {X 0,Y 271.618,Z 595.462,A -85,B 0,C 180,E1 -17863.18,E2 -17863.18} C_VEL
LIN {X 0,Y 270.585,Z 600.396,A -85,B 0,C 180,E1 -17864.947,E2 -17864.947} C_VEL
LIN {X 0,Y 269.533,Z 605.477,A -85,B 0,C 180,E1 -17867.316,E2 -17867.316} C_VEL
LIN {X 0,Y 268.914,Z 608.458,A -85,B 0,C 180,E1 -17869.28,E2 -17869.28} C_VEL
LIN {X 0,Y 268.297,Z 610.818,A -85,B 0,C 180,E1 -17871.799,E2 -17871.799} C_VEL
LIN {X 0,Y 268.106,Z 611.493,A -85,B 0,C 180,E1 -17872.92,E2 -17872.92} C_VEL
LIN {X 0,Y 267.926,Z 611.882,A -85,B 0,C 180,E1 -17874.753,E2 -17874.753} C_VEL
LIN {X 0,Y 267.87,Z 611.272,A -85,B 0,C 180,E1 -17877.095,E2 -17877.095} C_VEL
LIN {X 0,Y 267.975,Z 610.448,A -85,B 0,C 180,E1 -17878.363,E2 -17878.363} C_VEL
LIN {X 0,Y 268.257,Z 608.64,A -85,B 0,C 180,E1 -17880.146,E2 -17880.146} C_VEL
LIN {X 0,Y 268.574,Z 606.106,A -85,B 0,C 180,E1 -17881.899,E2 -17881.899} C_VEL
LIN {X 0,Y 268.935,Z 602.813,A -85,B 0,C 180,E1 -17883.623,E2 -17883.623} C_VEL
LIN {X 0,Y 269.629,Z 597.323,A -85,B 0,C 180,E1 -17885.824,E2 -17885.824} C_VEL
LIN {X 0,Y 270.318,Z 592.113,A -85,B 0,C 180,E1 -17887.449,E2 -17887.449} C_VEL
LIN {X 0,Y 271.243,Z 584.917,A -85,B 0,C 180,E1 -17889.25,E2 -17889.25} C_VEL
LIN {X 0,Y 272.089,Z 578.437,A -85,B 0,C 180,E1 -17890.575,E2 -17890.575} C_VEL
LIN {X 0,Y 272.978,Z 571.141,A -85,B 0,C 180,E1 -17891.809,E2 -17891.809} C_VEL
LIN {X 0,Y 273.837,Z 562.332,A -85,B 0,C 180,E1 -17893.025,E2 -17893.025} C_VEL
LIN {X 0,Y 272.756,Z 551.944,A -85,B 0,C 180,E1 -17894.245,E2 -17894.245} C_VEL
LIN {X 0,Y 271.104,Z 541.134,A -85,B 0,C 180,E1 -17895.212,E2 -17895.212} C_VEL
LIN {X 0,Y 269.465,Z 532.229,A -85,B 0,C 180,E1 -17895.826,E2 -17895.826} C_VEL
LIN {X 0,Y 269.212,Z 530.516,A -85,B 0,C 180,E1 -17895.984,E2 -17895.984} C_VEL
LIN {X 0,Y 269.592,Z 523.883,A -85,B 0,C 180,E1 -17900.243,E2 -17900.243} C_VEL
LIN {X 0,Y 270.015,Z 516.839,A -85,B 0,C 180,E1 -17904.772,E2 -17904.772} C_VEL
LIN {X 0,Y 270.342,Z 511.625,A -85,B 0,C 180,E1 -17908.23,E2 -17908.23} C_VEL
LIN {X 0,Y 270.755,Z 511.572,A -85,B 0,C 180,E1 -17909.999,E2 -17909.999} C_VEL
LIN {X 0,Y 270.633,Z 511.585,A -85,B 0,C 180,E1 -17912.976,E2 -17912.976} C_VEL
LIN {X 0,Y 270.613,Z 511.587,A -85,B 0,C 180,E1 -17917.46,E2 -17917.46} C_VEL
LIN {X 0,Y 270.443,Z 511.611,A -85,B 0,C 180,E1 -17920.48,E2 -17920.48} C_VEL
LIN {X 0,Y 270.404,Z 511.612,A -85,B 0,C 180,E1 -17925.064,E2 -17925.064} C_VEL
LIN {X 0,Y 270.302,Z 511.625,A -85,B 0,C 180,E1 -17929.755,E2 -17929.755} C_VEL
LIN {X 0,Y 270.274,Z 511.63,A -85,B 0,C 180,E1 -17934.585,E2 -17934.585} C_VEL
LIN {X 0,Y 270.274,Z 511.631,A -85,B 0,C 180,E1 -17937.907,E2 -17937.907} C_VEL
LIN {X 0,Y 270.184,Z 511.64,A -85,B 0,C 180,E1 -17941.347,E2 -17941.347} C_VEL
LIN {X 0,Y 270.214,Z 511.635,A -85,B 0,C 180,E1 -17944.903,E2 -17944.903} C_VEL
LIN {X 0,Y 270.221,Z 511.636,A -85,B 0,C 180,E1 -17948.716,E2 -17948.716} C_VEL
LIN {X 0,Y 270.199,Z 511.637,A -85,B 0,C 180,E1 -17952.552,E2 -17952.552} C_VEL
LIN {X 0,Y 270.212,Z 511.637,A -85,B 0,C 180,E1 -17956.739,E2 -17956.739} C_VEL
LIN {X 0,Y 270.244,Z 511.633,A -85,B 0,C 180,E1 -17959.447,E2 -17959.447} C_VEL
LIN {X 0,Y 270.256,Z 511.63,A -85,B 0,C 180,E1 -17963.721,E2 -17963.721} C_VEL
LIN {X 0,Y 270.202,Z 511.637,A -85,B 0,C 180,E1 -17966.892,E2 -17966.892} C_VEL
LIN {X 0,Y 270.194,Z 511.64,A -85,B 0,C 180,E1 -17970.382,E2 -17970.382} C_VEL
LIN {X 0,Y 270.261,Z 511.632,A -85,B 0,C 180,E1 -17973.763,E2 -17973.763} C_VEL
LIN {X 0,Y 270.23,Z 511.634,A -85,B 0,C 180,E1 -17977.038,E2 -17977.038} C_VEL
LIN {X 0,Y 270.299,Z 511.626,A -85,B 0,C 180,E1 -17980.244,E2 -17980.244} C_VEL
LIN {X 0,Y 270.401,Z 511.613,A -85,B 0,C 180,E1 -17984.935,E2 -17984.935} C_VEL
LIN {X 0,Y 270.44,Z 511.608,A -85,B 0,C 180,E1 -17989.519,E2 -17989.519} C_VEL
LIN {X 0,Y 270.609,Z 511.587,A -85,B 0,C 180,E1 -17992.539,E2 -17992.539} C_VEL
LIN {X 0,Y 270.786,Z 511.561,A -85,B 0,C 180,E1 -17998.513,E2 -17998.513} C_VEL
LIN {X 0,Y 270.785,Z 511.566,A -85,B 0,C 180,E1 -18001.487,E2 -18001.487} C_VEL
LIN {X 0,Y 270.609,Z 511.589,A -85,B 0,C 180,E1 -18007.461,E2 -18007.461} C_VEL
LIN {X 0,Y 270.439,Z 511.608,A -85,B 0,C 180,E1 -18010.481,E2 -18010.481} C_VEL
LIN {X 0,Y 270.4,Z 511.614,A -85,B 0,C 180,E1 -18015.065,E2 -18015.065} C_VEL
LIN {X 0,Y 270.327,Z 511.62,A -85,B 0,C 180,E1 -18016.878,E2 -18016.878} C_VEL
LIN {X 0,Y 269.572,Z 511.719,A -85,B 0,C 180,E1 -18018.121,E2 -18018.121} C_VEL
LIN {X 0,Y 266.629,Z 512.084,A -85,B 0,C 180,E1 -18020.146,E2 -18020.146} C_VEL
LIN {X 0,Y 264.21,Z 512.388,A -85,B 0,C 180,E1 -18021.792,E2 -18021.792} C_VEL
LIN {X 0,Y 263.228,Z 512.509,A -85,B 0,C 180,E1 -18023.07,E2 -18023.07} C_VEL
LIN {X 0,Y 263.175,Z 512.517,A -85,B 0,C 180,E1 -18023.502,E2 -18023.502} C_VEL
LIN {X 0,Y 263.19,Z 512.513,A -85,B 0,C 180,E1 -18026.997,E2 -18026.997} C_VEL
LIN {X 0,Y 263.138,Z 512.52,A -85,B 0,C 180,E1 -18031.279,E2 -18031.279} C_VEL
LIN {X 0,Y 263.17,Z 512.514,A -85,B 0,C 180,E1 -18034.122,E2 -18034.122} C_VEL
LIN {X 0,Y 263.163,Z 512.516,A -85,B 0,C 180,E1 -18037.896,E2 -18037.896} C_VEL
LIN {X 0,Y 263.14,Z 512.52,A -85,B 0,C 180,E1 -18041.89,E2 -18041.89} C_VEL
LIN {X 0,Y 263.137,Z 512.519,A -85,B 0,C 180,E1 -18046.148,E2 -18046.148} C_VEL
LIN {X 0,Y 263.252,Z 512.504,A -85,B 0,C 180,E1 -18050.733,E2 -18050.733} C_VEL
LIN {X 0,Y 263.437,Z 512.568,A -85,B 0,C 180,E1 -18052.299,E2 -18052.299} C_VEL
LIN {X 0,Y 264.308,Z 517.65,A -85,B 0,C 180,E1 -18056.056,E2 -18056.056} C_VEL
LIN {X 0,Y 264.558,Z 520.677,A -85,B 0,C 180,E1 -18058.22,E2 -18058.22} C_VEL
LIN {X 0,Y 263.521,Z 526.581,A -85,B 0,C 180,E1 -18062.309,E2 -18062.309} C_VEL
LIN {X 0,Y 262.49,Z 533.635,A -85,B 0,C 180,E1 -18067.157,E2 -18067.157} C_VEL
LIN {X 0,Y 262.089,Z 537.249,A -85,B 0,C 180,E1 -18069.644,E2 -18069.644} C_VEL
LIN {X 0,Y 263.794,Z 551.388,A -85,B 0,C 180,E1 -18070.353,E2 -18070.353} C_VEL
LIN {X 0,Y 264.756,Z 561.683,A -85,B 0,C 180,E1 -18071.141,E2 -18071.141} C_VEL
LIN {X 0,Y 265.289,Z 570.071,A -85,B 0,C 180,E1 -18071.968,E2 -18071.968} C_VEL
LIN {X 0,Y 265.557,Z 579.116,A -85,B 0,C 180,E1 -18073.076,E2 -18073.076} C_VEL
LIN {X 0,Y 265.337,Z 585.735,A -85,B 0,C 180,E1 -18074.051,E2 -18074.051} C_VEL
LIN {X 0,Y 264.349,Z 593.357,A -85,B 0,C 180,E1 -18075.371,E2 -18075.371} C_VEL
LIN {X 0,Y 263.24,Z 602.115,A -85,B 0,C 180,E1 -18077.277,E2 -18077.277} C_VEL
LIN {X 0,Y 262.363,Z 608.854,A -85,B 0,C 180,E1 -18079.193,E2 -18079.193} C_VEL
LIN {X 0,Y 261.865,Z 613.28,A -85,B 0,C 180,E1 -18080.734,E2 -18080.734} C_VEL
LIN {X 0,Y 261.353,Z 618.457,A -85,B 0,C 180,E1 -18083.05,E2 -18083.05} C_VEL
LIN {X 0,Y 261.152,Z 622.229,A -85,B 0,C 180,E1 -18085.37,E2 -18085.37} C_VEL
LIN {X 0,Y 261.146,Z 623.931,A -85,B 0,C 180,E1 -18086.915,E2 -18086.915} C_VEL
LIN {X 0,Y 261.152,Z 625.108,A -85,B 0,C 180,E1 -18088.459,E2 -18088.459} C_VEL
LIN {X 0,Y 261.171,Z 625.786,A -85,B 0,C 180,E1 -18090.001,E2 -18090.001} C_VEL
LIN {X 0,Y 261.149,Z 625.978,A -85,B 0,C 180,E1 -18091.543,E2 -18091.543} C_VEL
LIN {X 0,Y 261.139,Z 625.62,A -85,B 0,C 180,E1 -18093.086,E2 -18093.086} C_VEL
LIN {X 0,Y 261.224,Z 624.029,A -85,B 0,C 180,E1 -18095.467,E2 -18095.467} C_VEL
LIN {X 0,Y 262.057,Z 619.656,A -85,B 0,C 180,E1 -18099.261,E2 -18099.261} C_VEL
LIN {X 0,Y 262.706,Z 618.155,A -85,B 0,C 180,E1 -18100.794,E2 -18100.794} C_VEL
LIN {X 0,Y 264.102,Z 614.99,A -85,B 0,C 180,E1 -18103.074,E2 -18103.074} C_VEL
LIN {X 0,Y 266.076,Z 610.67,A -85,B 0,C 180,E1 -18105.316,E2 -18105.316} C_VEL
LIN {X 0,Y 268.935,Z 604.009,A -85,B 0,C 180,E1 -18107.883,E2 -18107.883} C_VEL
LIN {X 0,Y 271.394,Z 597.968,A -85,B 0,C 180,E1 -18109.674,E2 -18109.674} C_VEL
LIN {X 0,Y 273.811,Z 591.048,A -85,B 0,C 180,E1 -18111.405,E2 -18111.405} C_VEL
LIN {X 0,Y 274.973,Z 586.165,A -85,B 0,C 180,E1 -18112.544,E2 -18112.544} C_VEL
LIN {X 0,Y 275.63,Z 579.426,A -85,B 0,C 180,E1 -18114.078,E2 -18114.078} C_VEL
LIN {X 0,Y 275.641,Z 571.312,A -85,B 0,C 180,E1 -18115.91,E2 -18115.91} C_VEL
LIN {X 0,Y 274.338,Z 560.427,A -85,B 0,C 180,E1 -18118.467,E2 -18118.467} C_VEL
LIN {X 0,Y 272.395,Z 551.209,A -85,B 0,C 180,E1 -18120.841,E2 -18120.841} C_VEL
LIN {X 0,Y 271.202,Z 546.591,A -85,B 0,C 180,E1 -18122.135,E2 -18122.135} C_VEL
LIN {X 0,Y 270.092,Z 543.747,A -85,B 0,C 180,E1 -18123.124,E2 -18123.124} C_VEL
LIN {X 0,Y 269.34,Z 540.717,A -85,B 0,C 180,E1 -18124.046,E2 -18124.046} C_VEL
LIN {X 0,Y 267.41,Z 536.83,A -85,B 0,C 180,E1 -18125.814,E2 -18125.814} C_VEL
LIN {X 0,Y 266.772,Z 534.223,A -85,B 0,C 180,E1 -18126.823,E2 -18126.823} C_VEL
LIN {X 0,Y 266.602,Z 532.159,A -85,B 0,C 180,E1 -18130.139,E2 -18130.139} C_VEL
LIN {X 0,Y 266.393,Z 530.608,A -85,B 0,C 180,E1 -18133.31,E2 -18133.31} C_VEL
LIN {X 0,Y 266.185,Z 529.449,A -85,B 0,C 180,E1 -18136.649,E2 -18136.649} C_VEL
LIN {X 0,Y 266.016,Z 528.614,A -85,B 0,C 180,E1 -18140.649,E2 -18140.649} C_VEL
LIN {X 0,Y 265.959,Z 528.509,A -85,B 0,C 180,E1 -18142.869,E2 -18142.869} C_VEL
LIN {X 0,Y 267.344,Z 531.457,A -85,B 0,C 180,E1 -18144.666,E2 -18144.666} C_VEL
LIN {X 0,Y 269.478,Z 534.13,A -85,B 0,C 180,E1 -18146.571,E2 -18146.571} C_VEL
LIN {X 0,Y 271.87,Z 538.116,A -85,B 0,C 180,E1 -18148.548,E2 -18148.548} C_VEL
LIN {X 0,Y 272.939,Z 540.841,A -85,B 0,C 180,E1 -18149.613,E2 -18149.613} C_VEL
LIN {X 0,Y 275.666,Z 547.332,A -85,B 0,C 180,E1 -18151.998,E2 -18151.998} C_VEL
LIN {X 0,Y 278.004,Z 555.474,A -85,B 0,C 180,E1 -18154.548,E2 -18154.548} C_VEL
LIN {X 0,Y 279.119,Z 562.503,A -85,B 0,C 180,E1 -18156.583,E2 -18156.583} C_VEL
LIN {X 0,Y 279.15,Z 567.066,A -85,B 0,C 180,E1 -18157.812,E2 -18157.812} C_VEL
LIN {X 0,Y 276.239,Z 574.734,A -85,B 0,C 180,E1 -18159.524,E2 -18159.524} C_VEL
LIN {X 0,Y 272.983,Z 582.181,A -85,B 0,C 180,E1 -18161.616,E2 -18161.616} C_VEL
LIN {X 0,Y 270.59,Z 587.14,A -85,B 0,C 180,E1 -18163.399,E2 -18163.399} C_VEL
LIN {X 0,Y 268.06,Z 591.793,A -85,B 0,C 180,E1 -18165.578,E2 -18165.578} C_VEL
LIN {X 0,Y 265.783,Z 595.595,A -85,B 0,C 180,E1 -18168.066,E2 -18168.066} C_VEL
LIN {X 0,Y 263.689,Z 598.066,A -85,B 0,C 180,E1 -18170.798,E2 -18170.798} C_VEL
LIN {X 0,Y 262.958,Z 598.776,A -85,B 0,C 180,E1 -18172.321,E2 -18172.321} C_VEL
LIN {X 0,Y 262.483,Z 598.91,A -85,B 0,C 180,E1 -18173.852,E2 -18173.852} C_VEL
LIN {X 0,Y 262.017,Z 598.596,A -85,B 0,C 180,E1 -18175.385,E2 -18175.385} C_VEL
LIN {X 0,Y 261.627,Z 597.841,A -85,B 0,C 180,E1 -18176.92,E2 -18176.92} C_VEL
LIN {X 0,Y 261.353,Z 596.622,A -85,B 0,C 180,E1 -18178.459,E2 -18178.459} C_VEL
LIN {X 0,Y 261.221,Z 593.715,A -85,B 0,C 180,E1 -18180.771,E2 -18180.771} C_VEL
LIN {X 0,Y 261.378,Z 589.606,A -85,B 0,C 180,E1 -18183.083,E2 -18183.083} C_VEL
LIN {X 0,Y 261.441,Z 584.968,A -85,B 0,C 180,E1 -18185.065,E2 -18185.065} C_VEL
LIN {X 0,Y 261.832,Z 578.417,A -85,B 0,C 180,E1 -18187.286,E2 -18187.286} C_VEL
LIN {X 0,Y 262.292,Z 570.971,A -85,B 0,C 180,E1 -18189.252,E2 -18189.252} C_VEL
LIN {X 0,Y 262.817,Z 563.914,A -85,B 0,C 180,E1 -18190.789,E2 -18190.789} C_VEL
LIN {X 0,Y 263.457,Z 555.439,A -85,B 0,C 180,E1 -18192.322,E2 -18192.322} C_VEL
LIN {X 0,Y 264.218,Z 545.076,A -85,B 0,C 180,E1 -18193.851,E2 -18193.851} C_VEL
LIN {X 0,Y 264.426,Z 540.223,A -85,B 0,C 180,E1 -18194.429,E2 -18194.429} C_VEL
LIN {X 0,Y 262.744,Z 528.473,A -85,B 0,C 180,E1 -18195.644,E2 -18195.644} C_VEL
LIN {X 0,Y 261.541,Z 518.184,A -85,B 0,C 180,E1 -18196.438,E2 -18196.438} C_VEL
LIN {X 0,Y 261.612,Z 513.832,A -85,B 0,C 180,E1 -18200.852,E2 -18200.852} C_VEL
LIN {X 0,Y 263.52,Z 519.452,A -85,B 0,C 180,E1 -18204.935,E2 -18204.935} C_VEL
LIN {X 0,Y 264.141,Z 522.322,A -85,B 0,C 180,E1 -18206.893,E2 -18206.893} C_VEL
LIN {X 0,Y 263.753,Z 527.835,A -85,B 0,C 180,E1 -18210.416,E2 -18210.416} C_VEL
LIN {X 0,Y 263.507,Z 530.991,A -85,B 0,C 180,E1 -18212.406,E2 -18212.406} C_VEL
LIN {X 0,Y 266.395,Z 541.004,A -85,B 0,C 180,E1 -18213.36,E2 -18213.36} C_VEL
LIN {X 0,Y 268.525,Z 550.694,A -85,B 0,C 180,E1 -18214.432,E2 -18214.432} C_VEL
LIN {X 0,Y 269.955,Z 561.175,A -85,B 0,C 180,E1 -18215.77,E2 -18215.77} C_VEL
LIN {X 0,Y 270.29,Z 567.619,A -85,B 0,C 180,E1 -18216.73,E2 -18216.73} C_VEL
LIN {X 0,Y 268.617,Z 577.357,A -85,B 0,C 180,E1 -18218.287,E2 -18218.287} C_VEL
LIN {X 0,Y 267.195,Z 584.656,A -85,B 0,C 180,E1 -18219.762,E2 -18219.762} C_VEL
LIN {X 0,Y 265.786,Z 591.176,A -85,B 0,C 180,E1 -18221.381,E2 -18221.381} C_VEL
LIN {X 0,Y 264.623,Z 596.473,A -85,B 0,C 180,E1 -18223.002,E2 -18223.002} C_VEL
LIN {X 0,Y 263.446,Z 601.726,A -85,B 0,C 180,E1 -18225.012,E2 -18225.012} C_VEL
LIN {X 0,Y 262.546,Z 605.835,A -85,B 0,C 180,E1 -18227.066,E2 -18227.066} C_VEL
LIN {X 0,Y 261.972,Z 608.245,A -85,B 0,C 180,E1 -18228.691,E2 -18228.691} C_VEL
LIN {X 0,Y 261.317,Z 610.822,A -85,B 0,C 180,E1 -18231.255,E2 -18231.255} C_VEL
LIN {X 0,Y 260.886,Z 611.954,A -85,B 0,C 180,E1 -18233.918,E2 -18233.918} C_VEL
LIN {X 0,Y 260.754,Z 611.657,A -85,B 0,C 180,E1 -18236.671,E2 -18236.671} C_VEL
LIN {X 0,Y 261.04,Z 609.527,A -85,B 0,C 180,E1 -18239.49,E2 -18239.49} C_VEL
LIN {X 0,Y 261.453,Z 606.5,A -85,B 0,C 180,E1 -18241.812,E2 -18241.812} C_VEL
LIN {X 0,Y 261.863,Z 603.014,A -85,B 0,C 180,E1 -18243.714,E2 -18243.714} C_VEL
LIN {X 0,Y 262.562,Z 597.554,A -85,B 0,C 180,E1 -18245.965,E2 -18245.965} C_VEL
LIN {X 0,Y 263.274,Z 592.325,A -85,B 0,C 180,E1 -18247.641,E2 -18247.641} C_VEL
LIN {X 0,Y 264.234,Z 585.265,A -85,B 0,C 180,E1 -18249.458,E2 -18249.458} C_VEL
LIN {X 0,Y 265.109,Z 578.652,A -85,B 0,C 180,E1 -18250.848,E2 -18250.848} C_VEL
LIN {X 0,Y 266.086,Z 571.054,A -85,B 0,C 180,E1 -18252.161,E2 -18252.161} C_VEL
LIN {X 0,Y 266.867,Z 562.6,A -85,B 0,C 180,E1 -18253.357,E2 -18253.357} C_VEL
LIN {X 0,Y 265.685,Z 551.787,A -85,B 0,C 180,E1 -18254.661,E2 -18254.661} C_VEL
LIN {X 0,Y 264.06,Z 540.967,A -85,B 0,C 180,E1 -18255.649,E2 -18255.649} C_VEL
LIN {X 0,Y 262.18,Z 530.716,A -85,B 0,C 180,E1 -18256.385,E2 -18256.385} C_VEL
LIN {X 0,Y 262.513,Z 525.2,A -85,B 0,C 180,E1 -18259.978,E2 -18259.978} C_VEL
LIN {X 0,Y 262.877,Z 519.275,A -85,B 0,C 180,E1 -18263.86,E2 -18263.86} C_VEL
LIN {X 0,Y 263.325,Z 512.499,A -85,B 0,C 180,E1 -18268.374,E2 -18268.374} C_VEL
LIN {X 0,Y 263.714,Z 512.449,A -85,B 0,C 180,E1 -18269.999,E2 -18269.999} C_VEL
LIN {X 0,Y 263.754,Z 512.442,A -85,B 0,C 180,E1 -18271.526,E2 -18271.526} C_VEL
LIN {X 0,Y 263.574,Z 512.464,A -85,B 0,C 180,E1 -18277.661,E2 -18277.661} C_VEL
LIN {X 0,Y 263.375,Z 512.489,A -85,B 0,C 180,E1 -18280.765,E2 -18280.765} C_VEL
LIN {X 0,Y 263.352,Z 512.491,A -85,B 0,C 180,E1 -18285.477,E2 -18285.477} C_VEL
LIN {X 0,Y 263.264,Z 512.505,A -85,B 0,C 180,E1 -18290.306,E2 -18290.306} C_VEL
LIN {X 0,Y 263.209,Z 512.508,A -85,B 0,C 180,E1 -18295.29,E2 -18295.29} C_VEL
LIN {X 0,Y 263.183,Z 512.513,A -85,B 0,C 180,E1 -18298.728,E2 -18298.728} C_VEL
LIN {X 0,Y 263.133,Z 512.521,A -85,B 0,C 180,E1 -18302.287,E2 -18302.287} C_VEL
LIN {X 0,Y 263.186,Z 512.513,A -85,B 0,C 180,E1 -18305.977,E2 -18305.977} C_VEL
LIN {X 0,Y 263.131,Z 512.521,A -85,B 0,C 180,E1 -18309.867,E2 -18309.867} C_VEL
LIN {X 0,Y 263.142,Z 512.518,A -85,B 0,C 180,E1 -18313.979,E2 -18313.979} C_VEL
LIN {X 0,Y 263.172,Z 512.515,A -85,B 0,C 180,E1 -18318.394,E2 -18318.394} C_VEL
LIN {X 0,Y 263.187,Z 512.511,A -85,B 0,C 180,E1 -18322.108,E2 -18322.108} C_VEL
LIN {X 0,Y 263.181,Z 512.514,A -85,B 0,C 180,E1 -18325.89,E2 -18325.89} C_VEL
LIN {X 0,Y 263.139,Z 512.519,A -85,B 0,C 180,E1 -18329.505,E2 -18329.505} C_VEL
LIN {X 0,Y 263.19,Z 512.509,A -85,B 0,C 180,E1 -18333.002,E2 -18333.002} C_VEL
LIN {X 0,Y 263.182,Z 512.513,A -85,B 0,C 180,E1 -18336.387,E2 -18336.387} C_VEL
LIN {X 0,Y 263.261,Z 512.505,A -85,B 0,C 180,E1 -18339.693,E2 -18339.693} C_VEL
LIN {X 0,Y 263.349,Z 512.492,A -85,B 0,C 180,E1 -18344.522,E2 -18344.522} C_VEL
LIN {X 0,Y 263.372,Z 512.487,A -85,B 0,C 180,E1 -18349.234,E2 -18349.234} C_VEL
LIN {X 0,Y 263.57,Z 512.465,A -85,B 0,C 180,E1 -18352.338,E2 -18352.338} C_VEL
LIN {X 0,Y 263.75,Z 512.437,A -85,B 0,C 180,E1 -18358.473,E2 -18358.473} C_VEL
LIN {X 0,Y 263.75,Z 512.442,A -85,B 0,C 180,E1 -18361.527,E2 -18361.527} C_VEL
LIN {X 0,Y 263.57,Z 512.467,A -85,B 0,C 180,E1 -18367.662,E2 -18367.662} C_VEL
LIN {X 0,Y 263.371,Z 512.488,A -85,B 0,C 180,E1 -18370.766,E2 -18370.766} C_VEL
LIN {X 0,Y 263.348,Z 512.495,A -85,B 0,C 180,E1 -18375.478,E2 -18375.478} C_VEL
LIN {X 0,Y 263.261,Z 512.503,A -85,B 0,C 180,E1 -18380.307,E2 -18380.307} C_VEL
LIN {X 0,Y 263.175,Z 512.517,A -85,B 0,C 180,E1 -18383.502,E2 -18383.502} C_VEL
LIN {X 0,Y 262.574,Z 512.6,A -85,B 0,C 180,E1 -18384.78,E2 -18384.78} C_VEL
LIN {X 0,Y 259.72,Z 512.957,A -85,B 0,C 180,E1 -18386.862,E2 -18386.862} C_VEL
LIN {X 0,Y 257.243,Z 513.259,A -85,B 0,C 180,E1 -18388.556,E2 -18388.556} C_VEL
LIN {X 0,Y 256.164,Z 513.389,A -85,B 0,C 180,E1 -18389.871,E2 -18389.871} C_VEL
LIN {X 0,Y 256.07,Z 513.399,A -85,B 0,C 180,E1 -18390.317,E2 -18390.317} C_VEL
LIN {X 0,Y 256.121,Z 513.392,A -85,B 0,C 180,E1 -18394.595,E2 -18394.595} C_VEL
LIN {X 0,Y 256.126,Z 513.393,A -85,B 0,C 180,E1 -18397.275,E2 -18397.275} C_VEL
LIN {X 0,Y 256.072,Z 513.4,A -85,B 0,C 180,E1 -18401.2,E2 -18401.2} C_VEL
LIN {X 0,Y 256.068,Z 513.403,A -85,B 0,C 180,E1 -18405.528,E2 -18405.528} C_VEL
LIN {X 0,Y 256.187,Z 513.384,A -85,B 0,C 180,E1 -18410.186,E2 -18410.186} C_VEL
LIN {X 0,Y 256.411,Z 513.459,A -85,B 0,C 180,E1 -18412.415,E2 -18412.415} C_VEL
LIN {X 0,Y 257.448,Z 519.398,A -85,B 0,C 180,E1 -18416.91,E2 -18416.91} C_VEL
LIN {X 0,Y 257.35,Z 521.915,A -85,B 0,C 180,E1 -18418.744,E2 -18418.744} C_VEL
LIN {X 0,Y 256.203,Z 528.006,A -85,B 0,C 180,E1 -18423.089,E2 -18423.089} C_VEL
LIN {X 0,Y 255.341,Z 533.987,A -85,B 0,C 180,E1 -18427.336,E2 -18427.336} C_VEL
LIN {X 0,Y 255.06,Z 536.757,A -85,B 0,C 180,E1 -18429.159,E2 -18429.159} C_VEL
LIN {X 0,Y 256.814,Z 551.197,A -85,B 0,C 180,E1 -18429.916,E2 -18429.916} C_VEL
LIN {X 0,Y 257.785,Z 561.696,A -85,B 0,C 180,E1 -18430.749,E2 -18430.749} C_VEL
LIN {X 0,Y 258.333,Z 570.671,A -85,B 0,C 180,E1 -18431.672,E2 -18431.672} C_VEL
LIN {X 0,Y 258.589,Z 579.554,A -85,B 0,C 180,E1 -18432.81,E2 -18432.81} C_VEL
LIN {X 0,Y 258.341,Z 586.062,A -85,B 0,C 180,E1 -18433.81,E2 -18433.81} C_VEL
LIN {X 0,Y 257.176,Z 594.604,A -85,B 0,C 180,E1 -18435.359,E2 -18435.359} C_VEL
LIN {X 0,Y 256.082,Z 602.937,A -85,B 0,C 180,E1 -18437.318,E2 -18437.318} C_VEL
LIN {X 0,Y 255.369,Z 608.327,A -85,B 0,C 180,E1 -18438.894,E2 -18438.894} C_VEL
LIN {X 0,Y 254.844,Z 612.815,A -85,B 0,C 180,E1 -18440.477,E2 -18440.477} C_VEL
LIN {X 0,Y 254.424,Z 616.531,A -85,B 0,C 180,E1 -18442.062,E2 -18442.062} C_VEL
LIN {X 0,Y 254.18,Z 619.541,A -85,B 0,C 180,E1 -18443.651,E2 -18443.651} C_VEL
LIN {X 0,Y 254.061,Z 621.873,A -85,B 0,C 180,E1 -18445.24,E2 -18445.24} C_VEL
LIN {X 0,Y 254.061,Z 623.623,A -85,B 0,C 180,E1 -18446.829,E2 -18446.829} C_VEL
LIN {X 0,Y 254.08,Z 624.848,A -85,B 0,C 180,E1 -18448.416,E2 -18448.416} C_VEL
LIN {X 0,Y 254.096,Z 625.571,A -85,B 0,C 180,E1 -18450.001,E2 -18450.001} C_VEL
LIN {X 0,Y 254.055,Z 625.801,A -85,B 0,C 180,E1 -18451.586,E2 -18451.586} C_VEL
LIN {X 0,Y 254.036,Z 625.452,A -85,B 0,C 180,E1 -18453.173,E2 -18453.173} C_VEL
LIN {X 0,Y 254.125,Z 624.164,A -85,B 0,C 180,E1 -18455.376,E2 -18455.376} C_VEL
LIN {X 0,Y 255.038,Z 619.578,A -85,B 0,C 180,E1 -18459.518,E2 -18459.518} C_VEL
LIN {X 0,Y 255.741,Z 618.281,A -85,B 0,C 180,E1 -18461.092,E2 -18461.092} C_VEL
LIN {X 0,Y 257.206,Z 615.349,A -85,B 0,C 180,E1 -18463.431,E2 -18463.431} C_VEL
LIN {X 0,Y 259.274,Z 611.315,A -85,B 0,C 180,E1 -18465.728,E2 -18465.728} C_VEL
LIN {X 0,Y 262.265,Z 605.083,A -85,B 0,C 180,E1 -18468.354,E2 -18468.354} C_VEL
LIN {X 0,Y 265.427,Z 598.18,A -85,B 0,C 180,E1 -18470.539,E2 -18470.539} C_VEL
LIN {X 0,Y 267.968,Z 591.264,A -85,B 0,C 180,E1 -18472.353,E2 -18472.353} C_VEL
LIN {X 0,Y 269.378,Z 584.408,A -85,B 0,C 180,E1 -18474.057,E2 -18474.057} C_VEL
LIN {X 0,Y 269.884,Z 577.069,A -85,B 0,C 180,E1 -18475.861,E2 -18475.861} C_VEL
LIN {X 0,Y 269.713,Z 569.971,A -85,B 0,C 180,E1 -18477.632,E2 -18477.632} C_VEL
LIN {X 0,Y 268.843,Z 561.666,A -85,B 0,C 180,E1 -18479.782,E2 -18479.782} C_VEL
LIN {X 0,Y 267.562,Z 555.082,A -85,B 0,C 180,E1 -18481.692,E2 -18481.692} C_VEL
LIN {X 0,Y 267.003,Z 551.949,A -85,B 0,C 180,E1 -18482.617,E2 -18482.617} C_VEL
LIN {X 0,Y 265.339,Z 545.779,A -85,B 0,C 180,E1 -18484.806,E2 -18484.806} C_VEL
LIN {X 0,Y 263.949,Z 542.524,A -85,B 0,C 180,E1 -18486.331,E2 -18486.331} C_VEL
LIN {X 0,Y 263.704,Z 541.045,A -85,B 0,C 180,E1 -18486.915,E2 -18486.915} C_VEL
LIN {X 0,Y 262.067,Z 538.292,A -85,B 0,C 180,E1 -18488.949,E2 -18488.949} C_VEL
LIN {X 0,Y 260.379,Z 534.686,A -85,B 0,C 180,E1 -18492.438,E2 -18492.438} C_VEL
LIN {X 0,Y 260.006,Z 533.366,A -85,B 0,C 180,E1 -18494.652,E2 -18494.652} C_VEL
LIN {X 0,Y 260.093,Z 533.031,A -85,B 0,C 180,E1 -18496.851,E2 -18496.851} C_VEL
LIN {X 0,Y 261.804,Z 534.309,A -85,B 0,C 180,E1 -18501.124,E2 -18501.124} C_VEL
LIN {X 0,Y 262.432,Z 534.675,A -85,B 0,C 180,E1 -18501.979,E2 -18501.979} C_VEL
LIN {X 0,Y 265.03,Z 538.695,A -85,B 0,C 180,E1 -18505.292,E2 -18505.292} C_VEL
LIN {X 0,Y 266.911,Z 542.398,A -85,B 0,C 180,E1 -18507.416,E2 -18507.416} C_VEL
LIN {X 0,Y 269.047,Z 546.886,A -85,B 0,C 180,E1 -18509.546,E2 -18509.546} C_VEL
LIN {X 0,Y 271.061,Z 552.872,A -85,B 0,C 180,E1 -18511.831,E2 -18511.831} C_VEL
LIN {X 0,Y 272.745,Z 560.508,A -85,B 0,C 180,E1 -18514.406,E2 -18514.406} C_VEL
LIN {X 0,Y 273.373,Z 566.034,A -85,B 0,C 180,E1 -18516.124,E2 -18516.124} C_VEL
LIN {X 0,Y 273.345,Z 568.644,A -85,B 0,C 180,E1 -18516.925,E2 -18516.925} C_VEL
LIN {X 0,Y 272.394,Z 571.638,A -85,B 0,C 180,E1 -18517.632,E2 -18517.632} C_VEL
LIN {X 0,Y 269.326,Z 578.518,A -85,B 0,C 180,E1 -18519.373,E2 -18519.373} C_VEL
LIN {X 0,Y 266.478,Z 584.202,A -85,B 0,C 180,E1 -18521.151,E2 -18521.151} C_VEL
LIN {X 0,Y 263.97,Z 588.808,A -85,B 0,C 180,E1 -18522.971,E2 -18522.971} C_VEL
LIN {X 0,Y 261.34,Z 593.208,A -85,B 0,C 180,E1 -18525.198,E2 -18525.198} C_VEL
LIN {X 0,Y 259.012,Z 596.571,A -85,B 0,C 180,E1 -18527.642,E2 -18527.642} C_VEL
LIN {X 0,Y 256.734,Z 598.766,A -85,B 0,C 180,E1 -18530.547,E2 -18530.547} C_VEL
LIN {X 0,Y 255.967,Z 599.295,A -85,B 0,C 180,E1 -18532.109,E2 -18532.109} C_VEL
LIN {X 0,Y 255.45,Z 599.37,A -85,B 0,C 180,E1 -18533.682,E2 -18533.682} C_VEL
LIN {X 0,Y 254.965,Z 598.878,A -85,B 0,C 180,E1 -18535.257,E2 -18535.257} C_VEL
LIN {X 0,Y 254.561,Z 597.927,A -85,B 0,C 180,E1 -18536.835,E2 -18536.835} C_VEL
LIN {X 0,Y 254.279,Z 596.528,A -85,B 0,C 180,E1 -18538.416,E2 -18538.416} C_VEL
LIN {X 0,Y 254.146,Z 593.412,A -85,B 0,C 180,E1 -18540.792,E2 -18540.792} C_VEL
LIN {X 0,Y 254.312,Z 589.087,A -85,B 0,C 180,E1 -18543.169,E2 -18543.169} C_VEL
LIN {X 0,Y 254.467,Z 582.381,A -85,B 0,C 180,E1 -18545.871,E2 -18545.871} C_VEL
LIN {X 0,Y 254.955,Z 575.806,A -85,B 0,C 180,E1 -18547.922,E2 -18547.922} C_VEL
LIN {X 0,Y 255.292,Z 569.605,A -85,B 0,C 180,E1 -18549.508,E2 -18549.508} C_VEL
LIN {X 0,Y 255.813,Z 562.239,A -85,B 0,C 180,E1 -18551.088,E2 -18551.088} C_VEL
LIN {X 0,Y 256.646,Z 552.175,A -85,B 0,C 180,E1 -18552.856,E2 -18552.856} C_VEL
LIN {X 0,Y 257.303,Z 542.149,A -85,B 0,C 180,E1 -18554.231,E2 -18554.231} C_VEL
LIN {X 0,Y 256.852,Z 537.433,A -85,B 0,C 180,E1 -18554.803,E2 -18554.803} C_VEL
LIN {X 0,Y 255.34,Z 526.714,A -85,B 0,C 180,E1 -18555.849,E2 -18555.849} C_VEL
LIN {X 0,Y 254.455,Z 518.479,A -85,B 0,C 180,E1 -18556.549,E2 -18556.549} C_VEL
LIN {X 0,Y 254.522,Z 514.899,A -85,B 0,C 180,E1 -18560.246,E2 -18560.246} C_VEL
LIN {X 0,Y 256.327,Z 520.31,A -85,B 0,C 180,E1 -18564.285,E2 -18564.285} C_VEL
LIN {X 0,Y 257.223,Z 523.808,A -85,B 0,C 180,E1 -18566.797,E2 -18566.797} C_VEL
LIN {X 0,Y 256.787,Z 529.381,A -85,B 0,C 180,E1 -18570.42,E2 -18570.42} C_VEL
LIN {X 0,Y 256.686,Z 531.292,A -85,B 0,C 180,E1 -18571.574,E2 -18571.574} C_VEL
LIN {X 0,Y 259.49,Z 540.774,A -85,B 0,C 180,E1 -18572.521,E2 -18572.521} C_VEL
LIN {X 0,Y 261.558,Z 549.38,A -85,B 0,C 180,E1 -18573.516,E2 -18573.516} C_VEL
LIN {X 0,Y 262.861,Z 557.936,A -85,B 0,C 180,E1 -18574.622,E2 -18574.622} C_VEL
LIN {X 0,Y 263.647,Z 566.553,A -85,B 0,C 180,E1 -18575.906,E2 -18575.906} C_VEL
LIN {X 0,Y 263.326,Z 570.532,A -85,B 0,C 180,E1 -18576.515,E2 -18576.515} C_VEL
LIN {X 0,Y 261.811,Z 578.665,A -85,B 0,C 180,E1 -18577.915,E2 -18577.915} C_VEL
LIN {X 0,Y 260.346,Z 585.682,A -85,B 0,C 180,E1 -18579.4,E2 -18579.4} C_VEL
LIN {X 0,Y 258.854,Z 592.248,A -85,B 0,C 180,E1 -18581.111,E2 -18581.111} C_VEL
LIN {X 0,Y 257.478,Z 598.145,A -85,B 0,C 180,E1 -18583.031,E2 -18583.031} C_VEL
LIN {X 0,Y 256.108,Z 603.849,A -85,B 0,C 180,E1 -18585.519,E2 -18585.519} C_VEL
LIN {X 0,Y 255.324,Z 607.06,A -85,B 0,C 180,E1 -18587.387,E2 -18587.387} C_VEL
LIN {X 0,Y 254.931,Z 608.724,A -85,B 0,C 180,E1 -18588.574,E2 -18588.574} C_VEL
LIN {X 0,Y 254.34,Z 610.82,A -85,B 0,C 180,E1 -18590.688,E2 -18590.688} C_VEL
LIN {X 0,Y 253.971,Z 611.873,A -85,B 0,C 180,E1 -18592.497,E2 -18592.497} C_VEL
LIN {X 0,Y 253.739,Z 612.27,A -85,B 0,C 180,E1 -18594.432,E2 -18594.432} C_VEL
LIN {X 0,Y 253.665,Z 611.922,A -85,B 0,C 180,E1 -18596.349,E2 -18596.349} C_VEL
LIN {X 0,Y 253.872,Z 610.091,A -85,B 0,C 180,E1 -18599.113,E2 -18599.113} C_VEL
LIN {X 0,Y 254.253,Z 607.84,A -85,B 0,C 180,E1 -18601.07,E2 -18601.07} C_VEL
LIN {X 0,Y 254.572,Z 604.83,A -85,B 0,C 180,E1 -18602.964,E2 -18602.964} C_VEL
LIN {X 0,Y 255.233,Z 599.777,A -85,B 0,C 180,E1 -18605.323,E2 -18605.323} C_VEL
LIN {X 0,Y 255.988,Z 594.016,A -85,B 0,C 180,E1 -18607.395,E2 -18607.395} C_VEL
LIN {X 0,Y 256.912,Z 587.769,A -85,B 0,C 180,E1 -18609.168,E2 -18609.168} C_VEL
LIN {X 0,Y 257.989,Z 579.98,A -85,B 0,C 180,E1 -18610.919,E2 -18610.919} C_VEL
LIN {X 0,Y 258.888,Z 573.401,A -85,B 0,C 180,E1 -18612.137,E2 -18612.137} C_VEL
LIN {X 0,Y 259.761,Z 565.873,A -85,B 0,C 180,E1 -18613.293,E2 -18613.293} C_VEL
LIN {X 0,Y 259.797,Z 561.524,A -85,B 0,C 180,E1 -18613.901,E2 -18613.901} C_VEL
LIN {X 0,Y 258.495,Z 550.258,A -85,B 0,C 180,E1 -18615.232,E2 -18615.232} C_VEL
LIN {X 0,Y 257.001,Z 540.897,A -85,B 0,C 180,E1 -18616.105,E2 -18616.105} C_VEL
LIN {X 0,Y 255.265,Z 531.629,A -85,B 0,C 180,E1 -18616.769,E2 -18616.769} C_VEL
LIN {X 0,Y 255.173,Z 530.802,A -85,B 0,C 180,E1 -18616.866,E2 -18616.866} C_VEL
LIN {X 0,Y 255.506,Z 525.332,A -85,B 0,C 180,E1 -18620.5,E2 -18620.5} C_VEL
LIN {X 0,Y 255.921,Z 519.337,A -85,B 0,C 180,E1 -18624.484,E2 -18624.484} C_VEL
LIN {X 0,Y 256.381,Z 513.364,A -85,B 0,C 180,E1 -18628.625,E2 -18628.625} C_VEL
LIN {X 0,Y 256.672,Z 513.327,A -85,B 0,C 180,E1 -18629.999,E2 -18629.999} C_VEL
LIN {X 0,Y 256.717,Z 513.319,A -85,B 0,C 180,E1 -18631.568,E2 -18631.568} C_VEL
LIN {X 0,Y 256.542,Z 513.341,A -85,B 0,C 180,E1 -18637.872,E2 -18637.872} C_VEL
LIN {X 0,Y 256.311,Z 513.368,A -85,B 0,C 180,E1 -18641.065,E2 -18641.065} C_VEL
LIN {X 0,Y 256.301,Z 513.371,A -85,B 0,C 180,E1 -18645.914,E2 -18645.914} C_VEL
LIN {X 0,Y 256.167,Z 513.386,A -85,B 0,C 180,E1 -18650.894,E2 -18650.894} C_VEL
LIN {X 0,Y 256.189,Z 513.383,A -85,B 0,C 180,E1 -18655.138,E2 -18655.138} C_VEL
LIN {X 0,Y 256.116,Z 513.393,A -85,B 0,C 180,E1 -18659.598,E2 -18659.598} C_VEL
LIN {X 0,Y 256.084,Z 513.396,A -85,B 0,C 180,E1 -18663.289,E2 -18663.289} C_VEL
LIN {X 0,Y 256.128,Z 513.391,A -85,B 0,C 180,E1 -18667.274,E2 -18667.274} C_VEL
LIN {X 0,Y 256.081,Z 513.395,A -85,B 0,C 180,E1 -18671.197,E2 -18671.197} C_VEL
LIN {X 0,Y 256.074,Z 513.398,A -85,B 0,C 180,E1 -18674.473,E2 -18674.473} C_VEL
LIN {X 0,Y 256.102,Z 513.394,A -85,B 0,C 180,E1 -18678.806,E2 -18678.806} C_VEL
LIN {X 0,Y 256.154,Z 513.383,A -85,B 0,C 180,E1 -18682.871,E2 -18682.871} C_VEL
LIN {X 0,Y 256.083,Z 513.396,A -85,B 0,C 180,E1 -18686.709,E2 -18686.709} C_VEL
LIN {X 0,Y 256.125,Z 513.391,A -85,B 0,C 180,E1 -18691.409,E2 -18691.409} C_VEL
LIN {X 0,Y 256.165,Z 513.388,A -85,B 0,C 180,E1 -18695.699,E2 -18695.699} C_VEL
LIN {X 0,Y 256.164,Z 513.386,A -85,B 0,C 180,E1 -18699.105,E2 -18699.105} C_VEL
LIN {X 0,Y 256.298,Z 513.373,A -85,B 0,C 180,E1 -18704.085,E2 -18704.085} C_VEL
LIN {X 0,Y 256.308,Z 513.366,A -85,B 0,C 180,E1 -18708.934,E2 -18708.934} C_VEL
LIN {X 0,Y 256.538,Z 513.342,A -85,B 0,C 180,E1 -18712.127,E2 -18712.127} C_VEL
LIN {X 0,Y 256.713,Z 513.314,A -85,B 0,C 180,E1 -18718.431,E2 -18718.431} C_VEL
LIN {X 0,Y 256.713,Z 513.319,A -85,B 0,C 180,E1 -18721.569,E2 -18721.569} C_VEL
LIN {X 0,Y 256.538,Z 513.343,A -85,B 0,C 180,E1 -18727.873,E2 -18727.873} C_VEL
LIN {X 0,Y 256.307,Z 513.369,A -85,B 0,C 180,E1 -18731.066,E2 -18731.066} C_VEL
LIN {X 0,Y 256.297,Z 513.372,A -85,B 0,C 180,E1 -18735.915,E2 -18735.915} C_VEL
LIN {X 0,Y 256.166,Z 513.387,A -85,B 0,C 180,E1 -18740.895,E2 -18740.895} C_VEL
LIN {X 0,Y 256.186,Z 513.385,A -85,B 0,C 180,E1 -18745.139,E2 -18745.139} C_VEL
LIN {X 0,Y 256.108,Z 513.398,A -85,B 0,C 180,E1 -18749.6,E2 -18749.6} C_VEL
LIN {X 0,Y 256.07,Z 513.399,A -85,B 0,C 180,E1 -18750.317,E2 -18750.317} C_VEL
LIN {X 0,Y 255.387,Z 513.488,A -85,B 0,C 180,E1 -18751.631,E2 -18751.631} C_VEL
LIN {X 0,Y 252.535,Z 513.841,A -85,B 0,C 180,E1 -18753.773,E2 -18753.773} C_VEL
LIN {X 0,Y 250.133,Z 514.142,A -85,B 0,C 180,E1 -18755.516,E2 -18755.516} C_VEL
LIN {X 0,Y 249.116,Z 514.265,A -85,B 0,C 180,E1 -18756.868,E2 -18756.868} C_VEL
LIN {X 0,Y 249.04,Z 514.273,A -85,B 0,C 180,E1 -18757.326,E2 -18757.326} C_VEL
LIN {X 0,Y 249.029,Z 514.276,A -85,B 0,C 180,E1 -18760.473,E2 -18760.473} C_VEL
LIN {X 0,Y 249.012,Z 514.278,A -85,B 0,C 180,E1 -18764.877,E2 -18764.877} C_VEL
LIN {X 0,Y 249.047,Z 514.277,A -85,B 0,C 180,E1 -18767.371,E2 -18767.371} C_VEL
LIN {X 0,Y 249.373,Z 514.323,A -85,B 0,C 180,E1 -18772.535,E2 -18772.535} C_VEL
LIN {X 0,Y 250.299,Z 519.603,A -85,B 0,C 180,E1 -18776.653,E2 -18776.653} C_VEL
LIN {X 0,Y 250.259,Z 522.316,A -85,B 0,C 180,E1 -18778.7,E2 -18778.7} C_VEL
LIN {X 0,Y 249.107,Z 528.383,A -85,B 0,C 180,E1 -18783.167,E2 -18783.167} C_VEL
LIN {X 0,Y 248.21,Z 534.319,A -85,B 0,C 180,E1 -18787.528,E2 -18787.528} C_VEL
LIN {X 0,Y 248.074,Z 535.737,A -85,B 0,C 180,E1 -18788.461,E2 -18788.461} C_VEL
LIN {X 0,Y 248.128,Z 537.268,A -85,B 0,C 180,E1 -18788.721,E2 -18788.721} C_VEL
LIN {X 0,Y 249.849,Z 551.028,A -85,B 0,C 180,E1 -18789.464,E2 -18789.464} C_VEL
LIN {X 0,Y 250.759,Z 560.516,A -85,B 0,C 180,E1 -18790.225,E2 -18790.225} C_VEL
LIN {X 0,Y 251.3,Z 568.978,A -85,B 0,C 180,E1 -18791.092,E2 -18791.092} C_VEL
LIN {X 0,Y 251.559,Z 576.994,A -85,B 0,C 180,E1 -18792.103,E2 -18792.103} C_VEL
LIN {X 0,Y 251.585,Z 583.955,A -85,B 0,C 180,E1 -18793.153,E2 -18793.153} C_VEL
LIN {X 0,Y 250.636,Z 591.82,A -85,B 0,C 180,E1 -18794.552,E2 -18794.552} C_VEL
LIN {X 0,Y 249.555,Z 599.144,A -85,B 0,C 180,E1 -18796.151,E2 -18796.151} C_VEL
LIN {X 0,Y 248.551,Z 606.564,A -85,B 0,C 180,E1 -18798.171,E2 -18798.171} C_VEL
LIN {X 0,Y 247.832,Z 612.349,A -85,B 0,C 180,E1 -18800.204,E2 -18800.204} C_VEL
LIN {X 0,Y 247.383,Z 616.112,A -85,B 0,C 180,E1 -18801.835,E2 -18801.835} C_VEL
LIN {X 0,Y 247.118,Z 619.149,A -85,B 0,C 180,E1 -18803.469,E2 -18803.469} C_VEL
LIN {X 0,Y 246.969,Z 621.515,A -85,B 0,C 180,E1 -18805.103,E2 -18805.103} C_VEL
LIN {X 0,Y 246.959,Z 623.315,A -85,B 0,C 180,E1 -18806.738,E2 -18806.738} C_VEL
LIN {X 0,Y 246.987,Z 624.586,A -85,B 0,C 180,E1 -18808.37,E2 -18808.37} C_VEL
LIN {X 0,Y 247.023,Z 625.356,A -85,B 0,C 180,E1 -18810.001,E2 -18810.001} C_VEL
LIN {X 0,Y 246.963,Z 625.615,A -85,B 0,C 180,E1 -18811.632,E2 -18811.632} C_VEL
LIN {X 0,Y 246.937,Z 625.283,A -85,B 0,C 180,E1 -18813.264,E2 -18813.264} C_VEL
LIN {X 0,Y 247.022,Z 624.223,A -85,B 0,C 180,E1 -18815.265,E2 -18815.265} C_VEL
LIN {X 0,Y 247.505,Z 621.3,A -85,B 0,C 180,E1 -18818.163,E2 -18818.163} C_VEL
LIN {X 0,Y 248.037,Z 619.5,A -85,B 0,C 180,E1 -18819.789,E2 -18819.789} C_VEL
LIN {X 0,Y 248.775,Z 618.341,A -85,B 0,C 180,E1 -18821.406,E2 -18821.406} C_VEL
LIN {X 0,Y 250.327,Z 615.735,A -85,B 0,C 180,E1 -18823.807,E2 -18823.807} C_VEL
LIN {X 0,Y 252.491,Z 611.958,A -85,B 0,C 180,E1 -18826.162,E2 -18826.162} C_VEL
LIN {X 0,Y 255.138,Z 607.04,A -85,B 0,C 180,E1 -18828.469,E2 -18828.469} C_VEL
LIN {X 0,Y 257.661,Z 601.963,A -85,B 0,C 180,E1 -18830.352,E2 -18830.352} C_VEL
LIN {X 0,Y 260.615,Z 595.839,A -85,B 0,C 180,E1 -18832.182,E2 -18832.182} C_VEL
LIN {X 0,Y 262.528,Z 590.384,A -85,B 0,C 180,E1 -18833.676,E2 -18833.676} C_VEL
LIN {X 0,Y 263.599,Z 584.535,A -85,B 0,C 180,E1 -18835.252,E2 -18835.252} C_VEL
LIN {X 0,Y 264.242,Z 577.041,A -85,B 0,C 180,E1 -18837.247,E2 -18837.247} C_VEL
LIN {X 0,Y 263.866,Z 566.668,A -85,B 0,C 180,E1 -18840.135,E2 -18840.135} C_VEL
LIN {X 0,Y 262.667,Z 557.342,A -85,B 0,C 180,E1 -18843.034,E2 -18843.034} C_VEL
LIN {X 0,Y 261.591,Z 551.979,A -85,B 0,C 180,E1 -18844.995,E2 -18844.995} C_VEL
LIN {X 0,Y 260.255,Z 547.105,A -85,B 0,C 180,E1 -18847.288,E2 -18847.288} C_VEL
LIN {X 0,Y 259.339,Z 545.237,A -85,B 0,C 180,E1 -18848.558,E2 -18848.558} C_VEL
LIN {X 0,Y 258.032,Z 542.735,A -85,B 0,C 180,E1 -18850.821,E2 -18850.821} C_VEL
LIN {X 0,Y 257.389,Z 540.78,A -85,B 0,C 180,E1 -18853.05,E2 -18853.05} C_VEL
LIN {X 0,Y 257.202,Z 539.675,A -85,B 0,C 180,E1 -18855.272,E2 -18855.272} C_VEL
LIN {X 0,Y 257.382,Z 539.58,A -85,B 0,C 180,E1 -18857.499,E2 -18857.499} C_VEL
LIN {X 0,Y 259.336,Z 541.054,A -85,B 0,C 180,E1 -18861.805,E2 -18861.805} C_VEL
LIN {X 0,Y 261.259,Z 544.532,A -85,B 0,C 180,E1 -18864.942,E2 -18864.942} C_VEL
LIN {X 0,Y 263.434,Z 549.24,A -85,B 0,C 180,E1 -18867.753,E2 -18867.753} C_VEL
LIN {X 0,Y 264.956,Z 553.47,A -85,B 0,C 180,E1 -18869.737,E2 -18869.737} C_VEL
LIN {X 0,Y 266.192,Z 558.113,A -85,B 0,C 180,E1 -18871.625,E2 -18871.625} C_VEL
LIN {X 0,Y 267.231,Z 564.154,A -85,B 0,C 180,E1 -18873.839,E2 -18873.839} C_VEL
LIN {X 0,Y 267.525,Z 570.392,A -85,B 0,C 180,E1 -18875.972,E2 -18875.972} C_VEL
LIN {X 0,Y 267.435,Z 571.695,A -85,B 0,C 180,E1 -18876.374,E2 -18876.374} C_VEL
LIN {X 0,Y 264.227,Z 578.521,A -85,B 0,C 180,E1 -18878.138,E2 -18878.138} C_VEL
LIN {X 0,Y 260.564,Z 585.231,A -85,B 0,C 180,E1 -18880.297,E2 -18880.297} C_VEL
LIN {X 0,Y 257.385,Z 590.585,A -85,B 0,C 180,E1 -18882.521,E2 -18882.521} C_VEL
LIN {X 0,Y 254.611,Z 594.597,A -85,B 0,C 180,E1 -18884.798,E2 -18884.798} C_VEL
LIN {X 0,Y 252.152,Z 597.545,A -85,B 0,C 180,E1 -18887.3,E2 -18887.3} C_VEL
LIN {X 0,Y 251.028,Z 598.721,A -85,B 0,C 180,E1 -18888.698,E2 -18888.698} C_VEL
LIN {X 0,Y 249.771,Z 599.495,A -85,B 0,C 180,E1 -18890.281,E2 -18890.281} C_VEL
LIN {X 0,Y 248.957,Z 599.793,A -85,B 0,C 180,E1 -18891.886,E2 -18891.886} C_VEL
LIN {X 0,Y 248.4,Z 599.679,A -85,B 0,C 180,E1 -18893.502,E2 -18893.502} C_VEL
LIN {X 0,Y 247.916,Z 599.121,A -85,B 0,C 180,E1 -18895.122,E2 -18895.122} C_VEL
LIN {X 0,Y 247.497,Z 597.991,A -85,B 0,C 180,E1 -18896.744,E2 -18896.744} C_VEL
LIN {X 0,Y 247.124,Z 595.481,A -85,B 0,C 180,E1 -18899.185,E2 -18899.185} C_VEL
LIN {X 0,Y 247.107,Z 591.735,A -85,B 0,C 180,E1 -18901.63,E2 -18901.63} C_VEL
LIN {X 0,Y 247.247,Z 588.534,A -85,B 0,C 180,E1 -18903.259,E2 -18903.259} C_VEL
LIN {X 0,Y 247.342,Z 582.796,A -85,B 0,C 180,E1 -18905.556,E2 -18905.556} C_VEL
LIN {X 0,Y 247.837,Z 575.96,A -85,B 0,C 180,E1 -18907.741,E2 -18907.741} C_VEL
LIN {X 0,Y 248.286,Z 568.103,A -85,B 0,C 180,E1 -18909.778,E2 -18909.778} C_VEL
LIN {X 0,Y 249.041,Z 558.238,A -85,B 0,C 180,E1 -18911.806,E2 -18911.806} C_VEL
LIN {X 0,Y 249.685,Z 549.727,A -85,B 0,C 180,E1 -18913.221,E2 -18913.221} C_VEL
LIN {X 0,Y 250.205,Z 540.772,A -85,B 0,C 180,E1 -18914.436,E2 -18914.436} C_VEL
LIN {X 0,Y 248.657,Z 530.251,A -85,B 0,C 180,E1 -18915.604,E2 -18915.604} C_VEL
LIN {X 0,Y 247.381,Z 518.867,A -85,B 0,C 180,E1 -18916.558,E2 -18916.558} C_VEL
LIN {X 0,Y 247.424,Z 516.034,A -85,B 0,C 180,E1 -18919.605,E2 -18919.605} C_VEL
LIN {X 0,Y 249.392,Z 521.872,A -85,B 0,C 180,E1 -18924.118,E2 -18924.118} C_VEL
LIN {X 0,Y 250.306,Z 525.367,A -85,B 0,C 180,E1 -18926.695,E2 -18926.695} C_VEL
LIN {X 0,Y 249.836,Z 531.393,A -85,B 0,C 180,E1 -18930.655,E2 -18930.655} C_VEL
LIN {X 0,Y 252.925,Z 541.524,A -85,B 0,C 180,E1 -18931.75,E2 -18931.75} C_VEL
LIN {X 0,Y 254.91,Z 549.918,A -85,B 0,C 180,E1 -18932.767,E2 -18932.767} C_VEL
LIN {X 0,Y 256.293,Z 558.493,A -85,B 0,C 180,E1 -18933.933,E2 -18933.933} C_VEL
LIN {X 0,Y 257.029,Z 567.243,A -85,B 0,C 180,E1 -18935.288,E2 -18935.288} C_VEL
LIN {X 0,Y 256.85,Z 570.802,A -85,B 0,C 180,E1 -18935.871,E2 -18935.871} C_VEL
LIN {X 0,Y 255.3,Z 578.757,A -85,B 0,C 180,E1 -18937.274,E2 -18937.274} C_VEL
LIN {X 0,Y 253.712,Z 585.9,A -85,B 0,C 180,E1 -18938.822,E2 -18938.822} C_VEL
LIN {X 0,Y 252.131,Z 592.53,A -85,B 0,C 180,E1 -18940.599,E2 -18940.599} C_VEL
LIN {X 0,Y 250.298,Z 599.758,A -85,B 0,C 180,E1 -18943.109,E2 -18943.109} C_VEL
LIN {X 0,Y 249.188,Z 604.17,A -85,B 0,C 180,E1 -18945.162,E2 -18945.162} C_VEL
LIN {X 0,Y 248.207,Z 607.802,A -85,B 0,C 180,E1 -18947.408,E2 -18947.408} C_VEL
LIN {X 0,Y 247.613,Z 609.947,A -85,B 0,C 180,E1 -18949.245,E2 -18949.245} C_VEL
LIN {X 0,Y 247.093,Z 611.515,A -85,B 0,C 180,E1 -18951.263,E2 -18951.263} C_VEL
LIN {X 0,Y 246.794,Z 612.295,A -85,B 0,C 180,E1 -18953.271,E2 -18953.271} C_VEL
LIN {X 0,Y 246.571,Z 612.219,A -85,B 0,C 180,E1 -18955.75,E2 -18955.75} C_VEL
LIN {X 0,Y 246.726,Z 610.644,A -85,B 0,C 180,E1 -18958.711,E2 -18958.711} C_VEL
LIN {X 0,Y 247.151,Z 608.029,A -85,B 0,C 180,E1 -18961.091,E2 -18961.091} C_VEL
LIN {X 0,Y 247.73,Z 603.397,A -85,B 0,C 180,E1 -18963.913,E2 -18963.913} C_VEL
LIN {X 0,Y 248.482,Z 597.957,A -85,B 0,C 180,E1 -18966.283,E2 -18966.283} C_VEL
LIN {X 0,Y 249.403,Z 591.456,A -85,B 0,C 180,E1 -18968.422,E2 -18968.422} C_VEL
LIN {X 0,Y 250.191,Z 586.084,A -85,B 0,C 180,E1 -18969.872,E2 -18969.872} C_VEL
LIN {X 0,Y 251.131,Z 579.478,A -85,B 0,C 180,E1 -18971.354,E2 -18971.354} C_VEL
LIN {X 0,Y 252.204,Z 571.728,A -85,B 0,C 180,E1 -18972.777,E2 -18972.777} C_VEL
LIN {X 0,Y 252.978,Z 564.518,A -85,B 0,C 180,E1 -18973.87,E2 -18973.87} C_VEL
LIN {X 0,Y 252.311,Z 557.232,A -85,B 0,C 180,E1 -18974.862,E2 -18974.862} C_VEL
LIN {X 0,Y 251.257,Z 548.69,A -85,B 0,C 180,E1 -18975.832,E2 -18975.832} C_VEL
LIN {X 0,Y 249.673,Z 538.914,A -85,B 0,C 180,E1 -18976.726,E2 -18976.726} C_VEL
LIN {X 0,Y 248.139,Z 530.97,A -85,B 0,C 180,E1 -18977.319,E2 -18977.319} C_VEL
LIN {X 0,Y 248.511,Z 525.46,A -85,B 0,C 180,E1 -18981.052,E2 -18981.052} C_VEL
LIN {X 0,Y 248.924,Z 519.409,A -85,B 0,C 180,E1 -18985.14,E2 -18985.14} C_VEL
LIN {X 0,Y 249.38,Z 514.236,A -85,B 0,C 180,E1 -18988.788,E2 -18988.788} C_VEL
LIN {X 0,Y 249.678,Z 514.196,A -85,B 0,C 180,E1 -18991.612,E2 -18991.612} C_VEL
LIN {X 0,Y 249.463,Z 514.225,A -85,B 0,C 180,E1 -18996.47,E2 -18996.47} C_VEL
LIN {X 0,Y 249.426,Z 514.227,A -85,B 0,C 180,E1 -18999.732,E2 -18999.732} C_VEL
LIN {X 0,Y 249.207,Z 514.254,A -85,B 0,C 180,E1 -19004.702,E2 -19004.702} C_VEL
LIN {X 0,Y 249.14,Z 514.264,A -85,B 0,C 180,E1 -19008.076,E2 -19008.076} C_VEL
LIN {X 0,Y 249.087,Z 514.268,A -85,B 0,C 180,E1 -19011.517,E2 -19011.517} C_VEL
LIN {X 0,Y 249.131,Z 514.262,A -85,B 0,C 180,E1 -19015.482,E2 -19015.482} C_VEL
LIN {X 0,Y 249.086,Z 514.268,A -85,B 0,C 180,E1 -19018.994,E2 -19018.994} C_VEL
LIN {X 0,Y 249.035,Z 514.276,A -85,B 0,C 180,E1 -19022.424,E2 -19022.424} C_VEL
LIN {X 0,Y 249.068,Z 514.273,A -85,B 0,C 180,E1 -19026.338,E2 -19026.338} C_VEL
LIN {X 0,Y 249.034,Z 514.275,A -85,B 0,C 180,E1 -19030.471,E2 -19030.471} C_VEL
LIN {X 0,Y 249.045,Z 514.27,A -85,B 0,C 180,E1 -19032.801,E2 -19032.801} C_VEL
LIN {X 0,Y 249.061,Z 514.271,A -85,B 0,C 180,E1 -19037.372,E2 -19037.372} C_VEL
LIN {X 0,Y 249.051,Z 514.272,A -85,B 0,C 180,E1 -19041.624,E2 -19041.624} C_VEL
LIN {X 0,Y 249.06,Z 514.271,A -85,B 0,C 180,E1 -19045.642,E2 -19045.642} C_VEL
LIN {X 0,Y 249.046,Z 514.274,A -85,B 0,C 180,E1 -19049.472,E2 -19049.472} C_VEL
LIN {X 0,Y 249.07,Z 514.268,A -85,B 0,C 180,E1 -19053.162,E2 -19053.162} C_VEL
LIN {X 0,Y 249.077,Z 514.269,A -85,B 0,C 180,E1 -19056.732,E2 -19056.732} C_VEL
LIN {X 0,Y 249.108,Z 514.265,A -85,B 0,C 180,E1 -19060.211,E2 -19060.211} C_VEL
LIN {X 0,Y 249.239,Z 514.251,A -85,B 0,C 180,E1 -19063.622,E2 -19063.622} C_VEL
LIN {X 0,Y 249.251,Z 514.245,A -85,B 0,C 180,E1 -19068.616,E2 -19068.616} C_VEL
LIN {X 0,Y 249.482,Z 514.223,A -85,B 0,C 180,E1 -19071.903,E2 -19071.903} C_VEL
LIN {X 0,Y 249.435,Z 514.222,A -85,B 0,C 180,E1 -19076.769,E2 -19076.769} C_VEL
LIN {X 0,Y 249.726,Z 514.189,A -85,B 0,C 180,E1 -19080,E2 -19080} C_VEL
LIN {X 0,Y 249.436,Z 514.225,A -85,B 0,C 180,E1 -19083.23,E2 -19083.23} C_VEL
LIN {X 0,Y 249.482,Z 514.221,A -85,B 0,C 180,E1 -19088.097,E2 -19088.097} C_VEL
LIN {X 0,Y 249.25,Z 514.25,A -85,B 0,C 180,E1 -19091.383,E2 -19091.383} C_VEL
LIN {X 0,Y 249.239,Z 514.249,A -85,B 0,C 180,E1 -19096.378,E2 -19096.378} C_VEL
LIN {X 0,Y 249.085,Z 514.272,A -85,B 0,C 180,E1 -19101.518,E2 -19101.518} C_VEL
LIN {X 0,Y 249.128,Z 514.267,A -85,B 0,C 180,E1 -19105.482,E2 -19105.482} C_VEL
LIN {X 0,Y 249.078,Z 514.27,A -85,B 0,C 180,E1 -19108.993,E2 -19108.993} C_VEL
LIN {X 0,Y 249.034,Z 514.275,A -85,B 0,C 180,E1 -19112.425,E2 -19112.425} C_VEL
LIN {X 0,Y 249.066,Z 514.27,A -85,B 0,C 180,E1 -19116.339,E2 -19116.339} C_VEL
LIN {X 0,Y 249.04,Z 514.273,A -85,B 0,C 180,E1 -19117.326,E2 -19117.326} C_VEL
LIN {X 0,Y 248.385,Z 514.359,A -85,B 0,C 180,E1 -19118.676,E2 -19118.676} C_VEL
LIN {X 0,Y 245.522,Z 514.719,A -85,B 0,C 180,E1 -19120.877,E2 -19120.877} C_VEL
LIN {X 0,Y 243.075,Z 515.021,A -85,B 0,C 180,E1 -19122.669,E2 -19122.669} C_VEL
LIN {X 0,Y 242.018,Z 515.15,A -85,B 0,C 180,E1 -19124.06,E2 -19124.06} C_VEL
LIN {X 0,Y 241.929,Z 515.159,A -85,B 0,C 180,E1 -19124.532,E2 -19124.532} C_VEL
LIN {X 0,Y 241.977,Z 515.155,A -85,B 0,C 180,E1 -19128.087,E2 -19128.087} C_VEL
LIN {X 0,Y 242.346,Z 515.208,A -85,B 0,C 180,E1 -19132.71,E2 -19132.71} C_VEL
LIN {X 0,Y 243.256,Z 520.446,A -85,B 0,C 180,E1 -19136.913,E2 -19136.913} C_VEL
LIN {X 0,Y 243.178,Z 522.687,A -85,B 0,C 180,E1 -19138.655,E2 -19138.655} C_VEL
LIN {X 0,Y 241.984,Z 528.718,A -85,B 0,C 180,E1 -19143.246,E2 -19143.246} C_VEL
LIN {X 0,Y 241.081,Z 534.779,A -85,B 0,C 180,E1 -19147.731,E2 -19147.731} C_VEL
LIN {X 0,Y 241.126,Z 536.817,A -85,B 0,C 180,E1 -19148.211,E2 -19148.211} C_VEL
LIN {X 0,Y 242.911,Z 550.727,A -85,B 0,C 180,E1 -19148.989,E2 -19148.989} C_VEL
LIN {X 0,Y 243.782,Z 560.107,A -85,B 0,C 180,E1 -19149.761,E2 -19149.761} C_VEL
LIN {X 0,Y 244.36,Z 569.601,A -85,B 0,C 180,E1 -19150.774,E2 -19150.774} C_VEL
LIN {X 0,Y 244.609,Z 578.861,A -85,B 0,C 180,E1 -19152.015,E2 -19152.015} C_VEL
LIN {X 0,Y 244.373,Z 586.64,A -85,B 0,C 180,E1 -19153.287,E2 -19153.287} C_VEL
LIN {X 0,Y 243.152,Z 594.99,A -85,B 0,C 180,E1 -19154.923,E2 -19154.923} C_VEL
LIN {X 0,Y 241.977,Z 603.108,A -85,B 0,C 180,E1 -19156.993,E2 -19156.993} C_VEL
LIN {X 0,Y 241.047,Z 609.569,A -85,B 0,C 180,E1 -19159.076,E2 -19159.076} C_VEL
LIN {X 0,Y 240.571,Z 613.76,A -85,B 0,C 180,E1 -19160.755,E2 -19160.755} C_VEL
LIN {X 0,Y 240.179,Z 617.202,A -85,B 0,C 180,E1 -19162.434,E2 -19162.434} C_VEL
LIN {X 0,Y 239.899,Z 621.137,A -85,B 0,C 180,E1 -19164.959,E2 -19164.959} C_VEL
LIN {X 0,Y 239.86,Z 622.99,A -85,B 0,C 180,E1 -19166.641,E2 -19166.641} C_VEL
LIN {X 0,Y 239.896,Z 624.315,A -85,B 0,C 180,E1 -19168.322,E2 -19168.322} C_VEL
LIN {X 0,Y 239.952,Z 625.138,A -85,B 0,C 180,E1 -19170.001,E2 -19170.001} C_VEL
LIN {X 0,Y 239.873,Z 625.416,A -85,B 0,C 180,E1 -19171.68,E2 -19171.68} C_VEL
LIN {X 0,Y 239.842,Z 625.115,A -85,B 0,C 180,E1 -19173.361,E2 -19173.361} C_VEL
LIN {X 0,Y 239.912,Z 624.281,A -85,B 0,C 180,E1 -19175.128,E2 -19175.128} C_VEL
LIN {X 0,Y 240.108,Z 623.065,A -85,B 0,C 180,E1 -19176.724,E2 -19176.724} C_VEL
LIN {X 0,Y 240.729,Z 620.13,A -85,B 0,C 180,E1 -19179.241,E2 -19179.241} C_VEL
LIN {X 0,Y 240.963,Z 619.414,A -85,B 0,C 180,E1 -19179.867,E2 -19179.867} C_VEL
LIN {X 0,Y 241.81,Z 618.296,A -85,B 0,C 180,E1 -19181.74,E2 -19181.74} C_VEL
LIN {X 0,Y 242.834,Z 616.842,A -85,B 0,C 180,E1 -19183.388,E2 -19183.388} C_VEL
LIN {X 0,Y 244.939,Z 613.787,A -85,B 0,C 180,E1 -19185.819,E2 -19185.819} C_VEL
LIN {X 0,Y 247.512,Z 609.633,A -85,B 0,C 180,E1 -19188.201,E2 -19188.201} C_VEL
LIN {X 0,Y 251.113,Z 603.324,A -85,B 0,C 180,E1 -19190.907,E2 -19190.907} C_VEL
LIN {X 0,Y 254.255,Z 597.608,A -85,B 0,C 180,E1 -19192.768,E2 -19192.768} C_VEL
LIN {X 0,Y 256.333,Z 592.477,A -85,B 0,C 180,E1 -19194.285,E2 -19194.285} C_VEL
LIN {X 0,Y 257.872,Z 585.66,A -85,B 0,C 180,E1 -19196.288,E2 -19196.288} C_VEL
LIN {X 0,Y 258.576,Z 578.833,A -85,B 0,C 180,E1 -19198.272,E2 -19198.272} C_VEL
LIN {X 0,Y 258.625,Z 569.518,A -85,B 0,C 180,E1 -19201.086,E2 -19201.086} C_VEL
LIN {X 0,Y 258.047,Z 561.786,A -85,B 0,C 180,E1 -19203.704,E2 -19203.704} C_VEL
LIN {X 0,Y 257.3,Z 556.897,A -85,B 0,C 180,E1 -19205.667,E2 -19205.667} C_VEL
LIN {X 0,Y 256.033,Z 551.76,A -85,B 0,C 180,E1 -19208.404,E2 -19208.404} C_VEL
LIN {X 0,Y 254.516,Z 548.278,A -85,B 0,C 180,E1 -19211.793,E2 -19211.793} C_VEL
LIN {X 0,Y 254.149,Z 546.679,A -85,B 0,C 180,E1 -19214.03,E2 -19214.03} C_VEL
LIN {X 0,Y 254.119,Z 545.978,A -85,B 0,C 180,E1 -19216.259,E2 -19216.259} C_VEL
LIN {X 0,Y 254.412,Z 546.178,A -85,B 0,C 180,E1 -19218.472,E2 -19218.472} C_VEL
LIN {X 0,Y 255.286,Z 546.842,A -85,B 0,C 180,E1 -19220.714,E2 -19220.714} C_VEL
LIN {X 0,Y 256.397,Z 548.497,A -85,B 0,C 180,E1 -19222.913,E2 -19222.913} C_VEL
LIN {X 0,Y 257.616,Z 550.857,A -85,B 0,C 180,E1 -19225.048,E2 -19225.048} C_VEL
LIN {X 0,Y 259.289,Z 555.318,A -85,B 0,C 180,E1 -19227.79,E2 -19227.79} C_VEL
LIN {X 0,Y 260.628,Z 560.189,A -85,B 0,C 180,E1 -19230.169,E2 -19230.169} C_VEL
LIN {X 0,Y 261.579,Z 566.614,A -85,B 0,C 180,E1 -19232.823,E2 -19232.823} C_VEL
LIN {X 0,Y 261.769,Z 572.323,A -85,B 0,C 180,E1 -19234.985,E2 -19234.985} C_VEL
LIN {X 0,Y 261.387,Z 574.571,A -85,B 0,C 180,E1 -19235.793,E2 -19235.793} C_VEL
LIN {X 0,Y 257.337,Z 582.208,A -85,B 0,C 180,E1 -19237.944,E2 -19237.944} C_VEL
LIN {X 0,Y 254.162,Z 587.376,A -85,B 0,C 180,E1 -19239.779,E2 -19239.779} C_VEL
LIN {X 0,Y 250.799,Z 592.219,A -85,B 0,C 180,E1 -19242.047,E2 -19242.047} C_VEL
LIN {X 0,Y 247.897,Z 595.866,A -85,B 0,C 180,E1 -19244.376,E2 -19244.376} C_VEL
LIN {X 0,Y 245.301,Z 598.531,A -85,B 0,C 180,E1 -19246.94,E2 -19246.94} C_VEL
LIN {X 0,Y 242.822,Z 600.185,A -85,B 0,C 180,E1 -19250,E2 -19250} C_VEL
LIN {X 0,Y 241.954,Z 600.298,A -85,B 0,C 180,E1 -19251.649,E2 -19251.649} C_VEL
LIN {X 0,Y 241.355,Z 599.954,A -85,B 0,C 180,E1 -19253.311,E2 -19253.311} C_VEL
LIN {X 0,Y 240.848,Z 599.203,A -85,B 0,C 180,E1 -19254.978,E2 -19254.978} C_VEL
LIN {X 0,Y 240.436,Z 598.01,A -85,B 0,C 180,E1 -19256.649,E2 -19256.649} C_VEL
LIN {X 0,Y 240.051,Z 595.162,A -85,B 0,C 180,E1 -19259.161,E2 -19259.161} C_VEL
LIN {X 0,Y 240.039,Z 591.131,A -85,B 0,C 180,E1 -19261.678,E2 -19261.678} C_VEL
LIN {X 0,Y 240.176,Z 585.806,A -85,B 0,C 180,E1 -19264.195,E2 -19264.195} C_VEL
LIN {X 0,Y 240.478,Z 578.909,A -85,B 0,C 180,E1 -19266.713,E2 -19266.713} C_VEL
LIN {X 0,Y 240.977,Z 571.539,A -85,B 0,C 180,E1 -19268.808,E2 -19268.808} C_VEL
LIN {X 0,Y 241.456,Z 564.446,A -85,B 0,C 180,E1 -19270.482,E2 -19270.482} C_VEL
LIN {X 0,Y 242.076,Z 555.964,A -85,B 0,C 180,E1 -19272.151,E2 -19272.151} C_VEL
LIN {X 0,Y 242.851,Z 545.574,A -85,B 0,C 180,E1 -19273.813,E2 -19273.813} C_VEL
LIN {X 0,Y 243.041,Z 540.743,A -85,B 0,C 180,E1 -19274.443,E2 -19274.443} C_VEL
LIN {X 0,Y 241.27,Z 528.395,A -85,B 0,C 180,E1 -19275.801,E2 -19275.801} C_VEL
LIN {X 0,Y 240.301,Z 519.203,A -85,B 0,C 180,E1 -19276.603,E2 -19276.603} C_VEL
LIN {X 0,Y 240.274,Z 517.201,A -85,B 0,C 180,E1 -19278.88,E2 -19278.88} C_VEL
LIN {X 0,Y 242.081,Z 522.382,A -85,B 0,C 180,E1 -19283.075,E2 -19283.075} C_VEL
LIN {X 0,Y 243.361,Z 526.777,A -85,B 0,C 180,E1 -19286.458,E2 -19286.458} C_VEL
LIN {X 0,Y 243.015,Z 531.35,A -85,B 0,C 180,E1 -19289.598,E2 -19289.598} C_VEL
LIN {X 0,Y 244.992,Z 537.456,A -85,B 0,C 180,E1 -19290.318,E2 -19290.318} C_VEL
LIN {X 0,Y 247.834,Z 548.072,A -85,B 0,C 180,E1 -19291.644,E2 -19291.644} C_VEL
LIN {X 0,Y 249.384,Z 556.747,A -85,B 0,C 180,E1 -19292.854,E2 -19292.854} C_VEL
LIN {X 0,Y 250.245,Z 565.196,A -85,B 0,C 180,E1 -19294.173,E2 -19294.173} C_VEL
LIN {X 0,Y 250.468,Z 570.845,A -85,B 0,C 180,E1 -19295.151,E2 -19295.151} C_VEL
LIN {X 0,Y 248.789,Z 578.956,A -85,B 0,C 180,E1 -19296.609,E2 -19296.609} C_VEL
LIN {X 0,Y 247.117,Z 586.222,A -85,B 0,C 180,E1 -19298.227,E2 -19298.227} C_VEL
LIN {X 0,Y 245.472,Z 592.707,A -85,B 0,C 180,E1 -19300.009,E2 -19300.009} C_VEL
LIN {X 0,Y 243.843,Z 598.741,A -85,B 0,C 180,E1 -19302.083,E2 -19302.083} C_VEL
LIN {X 0,Y 242.634,Z 603.168,A -85,B 0,C 180,E1 -19304.041,E2 -19304.041} C_VEL
LIN {X 0,Y 241.368,Z 607.593,A -85,B 0,C 180,E1 -19306.714,E2 -19306.714} C_VEL
LIN {X 0,Y 240.97,Z 609.119,A -85,B 0,C 180,E1 -19307.87,E2 -19307.87} C_VEL
LIN {X 0,Y 240.316,Z 611.102,A -85,B 0,C 180,E1 -19309.954,E2 -19309.954} C_VEL
LIN {X 0,Y 239.808,Z 612.362,A -85,B 0,C 180,E1 -19312.306,E2 -19312.306} C_VEL
LIN {X 0,Y 239.59,Z 612.661,A -85,B 0,C 180,E1 -19314.078,E2 -19314.078} C_VEL
LIN {X 0,Y 239.484,Z 612.308,A -85,B 0,C 180,E1 -19316.11,E2 -19316.11} C_VEL
LIN {X 0,Y 239.588,Z 611.129,A -85,B 0,C 180,E1 -19318.286,E2 -19318.286} C_VEL
LIN {X 0,Y 239.844,Z 609.416,A -85,B 0,C 180,E1 -19320.122,E2 -19320.122} C_VEL
LIN {X 0,Y 240.245,Z 606.866,A -85,B 0,C 180,E1 -19322.091,E2 -19322.091} C_VEL
LIN {X 0,Y 240.85,Z 602.058,A -85,B 0,C 180,E1 -19324.767,E2 -19324.767} C_VEL
LIN {X 0,Y 241.605,Z 596.951,A -85,B 0,C 180,E1 -19326.877,E2 -19326.877} C_VEL
LIN {X 0,Y 242.427,Z 591.223,A -85,B 0,C 180,E1 -19328.772,E2 -19328.772} C_VEL
LIN {X 0,Y 243.197,Z 586.222,A -85,B 0,C 180,E1 -19330.149,E2 -19330.149} C_VEL
LIN {X 0,Y 244.216,Z 579.258,A -85,B 0,C 180,E1 -19331.744,E2 -19331.744} C_VEL
LIN {X 0,Y 245.29,Z 571.834,A -85,B 0,C 180,E1 -19333.135,E2 -19333.135} C_VEL
LIN {X 0,Y 246.003,Z 564.684,A -85,B 0,C 180,E1 -19334.251,E2 -19334.251} C_VEL
LIN {X 0,Y 245.14,Z 555.885,A -85,B 0,C 180,E1 -19335.471,E2 -19335.471} C_VEL
LIN {X 0,Y 243.704,Z 545.27,A -85,B 0,C 180,E1 -19336.661,E2 -19336.661} C_VEL
LIN {X 0,Y 241.602,Z 533.723,A -85,B 0,C 180,E1 -19337.611,E2 -19337.611} C_VEL
LIN {X 0,Y 241.151,Z 531.133,A -85,B 0,C 180,E1 -19337.801,E2 -19337.801} C_VEL
LIN {X 0,Y 241.543,Z 525.548,A -85,B 0,C 180,E1 -19341.634,E2 -19341.634} C_VEL
LIN {X 0,Y 241.974,Z 519.476,A -85,B 0,C 180,E1 -19345.835,E2 -19345.835} C_VEL
LIN {X 0,Y 242.376,Z 515.108,A -85,B 0,C 180,E1 -19348.961,E2 -19348.961} C_VEL
LIN {X 0,Y 242.639,Z 515.073,A -85,B 0,C 180,E1 -19351.659,E2 -19351.659} C_VEL
LIN {X 0,Y 242.436,Z 515.099,A -85,B 0,C 180,E1 -19356.658,E2 -19356.658} C_VEL
LIN {X 0,Y 242.347,Z 515.111,A -85,B 0,C 180,E1 -19360.02,E2 -19360.02} C_VEL
LIN {X 0,Y 242.168,Z 515.13,A -85,B 0,C 180,E1 -19365.14,E2 -19365.14} C_VEL
LIN {X 0,Y 242.074,Z 515.142,A -85,B 0,C 180,E1 -19368.623,E2 -19368.623} C_VEL
LIN {X 0,Y 242.013,Z 515.152,A -85,B 0,C 180,E1 -19372.179,E2 -19372.179} C_VEL
LIN {X 0,Y 242.066,Z 515.144,A -85,B 0,C 180,E1 -19375.837,E2 -19375.837} C_VEL
LIN {X 0,Y 242.031,Z 515.147,A -85,B 0,C 180,E1 -19379.579,E2 -19379.579} C_VEL
LIN {X 0,Y 241.991,Z 515.152,A -85,B 0,C 180,E1 -19383.49,E2 -19383.49} C_VEL
LIN {X 0,Y 242.003,Z 515.151,A -85,B 0,C 180,E1 -19387.578,E2 -19387.578} C_VEL
LIN {X 0,Y 241.966,Z 515.156,A -85,B 0,C 180,E1 -19391.915,E2 -19391.915} C_VEL
LIN {X 0,Y 241.99,Z 515.153,A -85,B 0,C 180,E1 -19396.556,E2 -19396.556} C_VEL
LIN {X 0,Y 242.006,Z 515.15,A -85,B 0,C 180,E1 -19400.291,E2 -19400.291} C_VEL
LIN {X 0,Y 242.035,Z 515.145,A -85,B 0,C 180,E1 -19404.497,E2 -19404.497} C_VEL
LIN {X 0,Y 241.973,Z 515.155,A -85,B 0,C 180,E1 -19408.479,E2 -19408.479} C_VEL
LIN {X 0,Y 242.001,Z 515.15,A -85,B 0,C 180,E1 -19412.312,E2 -19412.312} C_VEL
LIN {X 0,Y 242.055,Z 515.148,A -85,B 0,C 180,E1 -19416.016,E2 -19416.016} C_VEL
LIN {X 0,Y 242.035,Z 515.148,A -85,B 0,C 180,E1 -19419.608,E2 -19419.608} C_VEL
LIN {X 0,Y 242.161,Z 515.131,A -85,B 0,C 180,E1 -19423.278,E2 -19423.278} C_VEL
LIN {X 0,Y 242.185,Z 515.127,A -85,B 0,C 180,E1 -19428.28,E2 -19428.28} C_VEL
LIN {X 0,Y 242.433,Z 515.099,A -85,B 0,C 180,E1 -19431.666,E2 -19431.666} C_VEL
LIN {X 0,Y 242.26,Z 515.118,A -85,B 0,C 180,E1 -19435.007,E2 -19435.007} C_VEL
LIN {X 0,Y 242.635,Z 515.067,A -85,B 0,C 180,E1 -19438.34,E2 -19438.34} C_VEL
LIN {X 0,Y 242.635,Z 515.073,A -85,B 0,C 180,E1 -19441.66,E2 -19441.66} C_VEL
LIN {X 0,Y 242.432,Z 515.096,A -85,B 0,C 180,E1 -19446.659,E2 -19446.659} C_VEL
LIN {X 0,Y 242.343,Z 515.11,A -85,B 0,C 180,E1 -19450.02,E2 -19450.02} C_VEL
LIN {X 0,Y 242.164,Z 515.132,A -85,B 0,C 180,E1 -19455.141,E2 -19455.141} C_VEL
LIN {X 0,Y 242.071,Z 515.143,A -85,B 0,C 180,E1 -19458.624,E2 -19458.624} C_VEL
LIN {X 0,Y 242.011,Z 515.152,A -85,B 0,C 180,E1 -19462.18,E2 -19462.18} C_VEL
LIN {X 0,Y 242.064,Z 515.147,A -85,B 0,C 180,E1 -19465.838,E2 -19465.838} C_VEL
LIN {X 0,Y 242.027,Z 515.152,A -85,B 0,C 180,E1 -19469.58,E2 -19469.58} C_VEL
LIN {X 0,Y 241.989,Z 515.157,A -85,B 0,C 180,E1 -19473.491,E2 -19473.491} C_VEL
LIN {X 0,Y 242,Z 515.153,A -85,B 0,C 180,E1 -19477.58,E2 -19477.58} C_VEL
LIN {X 0,Y 241.95,Z 515.159,A -85,B 0,C 180,E1 -19481.92,E2 -19481.92} C_VEL
LIN {X 0,Y 241.929,Z 515.159,A -85,B 0,C 180,E1 -19484.532,E2 -19484.532} C_VEL
LIN {X 0,Y 241.248,Z 515.247,A -85,B 0,C 180,E1 -19485.921,E2 -19485.921} C_VEL
LIN {X 0,Y 238.407,Z 515.599,A -85,B 0,C 180,E1 -19488.189,E2 -19488.189} C_VEL
LIN {X 0,Y 236.083,Z 515.89,A -85,B 0,C 180,E1 -19490.037,E2 -19490.037} C_VEL
LIN {X 0,Y 235.2,Z 516.002,A -85,B 0,C 180,E1 -19491.47,E2 -19491.47} C_VEL
LIN {X 0,Y 235.188,Z 516.002,A -85,B 0,C 180,E1 -19491.954,E2 -19491.954} C_VEL
LIN {X 0,Y 235.292,Z 516.093,A -85,B 0,C 180,E1 -19492.917,E2 -19492.917} C_VEL
LIN {X 0,Y 236.078,Z 520.372,A -85,B 0,C 180,E1 -19496.465,E2 -19496.465} C_VEL
LIN {X 0,Y 236.1,Z 523.028,A -85,B 0,C 180,E1 -19498.607,E2 -19498.607} C_VEL
LIN {X 0,Y 234.875,Z 529.03,A -85,B 0,C 180,E1 -19503.332,E2 -19503.332} C_VEL
LIN {X 0,Y 234.116,Z 533.677,A -85,B 0,C 180,E1 -19506.914,E2 -19506.914} C_VEL
LIN {X 0,Y 234.159,Z 536.644,A -85,B 0,C 180,E1 -19507.663,E2 -19507.663} C_VEL
LIN {X 0,Y 236.023,Z 550.902,A -85,B 0,C 180,E1 -19508.523,E2 -19508.523} C_VEL
LIN {X 0,Y 236.878,Z 560.714,A -85,B 0,C 180,E1 -19509.372,E2 -19509.372} C_VEL
LIN {X 0,Y 237.382,Z 569.281,A -85,B 0,C 180,E1 -19510.321,E2 -19510.321} C_VEL
LIN {X 0,Y 237.648,Z 577.702,A -85,B 0,C 180,E1 -19511.474,E2 -19511.474} C_VEL
LIN {X 0,Y 237.523,Z 585.646,A -85,B 0,C 180,E1 -19512.79,E2 -19512.79} C_VEL
LIN {X 0,Y 236.3,Z 594.161,A -85,B 0,C 180,E1 -19514.475,E2 -19514.475} C_VEL
LIN {X 0,Y 235.025,Z 602.45,A -85,B 0,C 180,E1 -19516.601,E2 -19516.601} C_VEL
LIN {X 0,Y 234.245,Z 607.824,A -85,B 0,C 180,E1 -19518.317,E2 -19518.317} C_VEL
LIN {X 0,Y 233.532,Z 613.252,A -85,B 0,C 180,E1 -19520.474,E2 -19520.474} C_VEL
LIN {X 0,Y 233.125,Z 616.76,A -85,B 0,C 180,E1 -19522.204,E2 -19522.204} C_VEL
LIN {X 0,Y 232.812,Z 621.001,A -85,B 0,C 180,E1 -19524.991,E2 -19524.991} C_VEL
LIN {X 0,Y 232.766,Z 622.665,A -85,B 0,C 180,E1 -19526.539,E2 -19526.539} C_VEL
LIN {X 0,Y 232.807,Z 624.044,A -85,B 0,C 180,E1 -19528.271,E2 -19528.271} C_VEL
LIN {X 0,Y 232.882,Z 624.916,A -85,B 0,C 180,E1 -19530.001,E2 -19530.001} C_VEL
LIN {X 0,Y 232.785,Z 625.204,A -85,B 0,C 180,E1 -19531.731,E2 -19531.731} C_VEL
LIN {X 0,Y 232.751,Z 624.948,A -85,B 0,C 180,E1 -19533.463,E2 -19533.463} C_VEL
LIN {X 0,Y 232.84,Z 624.218,A -85,B 0,C 180,E1 -19535.196,E2 -19535.196} C_VEL
LIN {X 0,Y 233.059,Z 623.008,A -85,B 0,C 180,E1 -19536.929,E2 -19536.929} C_VEL
LIN {X 0,Y 233.729,Z 620.139,A -85,B 0,C 180,E1 -19539.52,E2 -19539.52} C_VEL
LIN {X 0,Y 234.038,Z 619.071,A -85,B 0,C 180,E1 -19540.381,E2 -19540.381} C_VEL
LIN {X 0,Y 235.939,Z 617.057,A -85,B 0,C 180,E1 -19543.787,E2 -19543.787} C_VEL
LIN {X 0,Y 238.152,Z 614.276,A -85,B 0,C 180,E1 -19546.282,E2 -19546.282} C_VEL
LIN {X 0,Y 240.82,Z 610.422,A -85,B 0,C 180,E1 -19548.726,E2 -19548.726} C_VEL
LIN {X 0,Y 243.967,Z 605.468,A -85,B 0,C 180,E1 -19551.107,E2 -19551.107} C_VEL
LIN {X 0,Y 247.882,Z 599.184,A -85,B 0,C 180,E1 -19553.387,E2 -19553.387} C_VEL
LIN {X 0,Y 250.55,Z 593.228,A -85,B 0,C 180,E1 -19555.32,E2 -19555.32} C_VEL
LIN {X 0,Y 252.173,Z 586.724,A -85,B 0,C 180,E1 -19557.377,E2 -19557.377} C_VEL
LIN {X 0,Y 253.007,Z 580.646,A -85,B 0,C 180,E1 -19559.329,E2 -19559.329} C_VEL
LIN {X 0,Y 253.437,Z 572.077,A -85,B 0,C 180,E1 -19562.208,E2 -19562.208} C_VEL
LIN {X 0,Y 253.173,Z 564.998,A -85,B 0,C 180,E1 -19564.898,E2 -19564.898} C_VEL
LIN {X 0,Y 252.929,Z 561.831,A -85,B 0,C 180,E1 -19566.312,E2 -19566.312} C_VEL
LIN {X 0,Y 252.157,Z 557.562,A -85,B 0,C 180,E1 -19568.703,E2 -19568.703} C_VEL
LIN {X 0,Y 250.902,Z 554.155,A -85,B 0,C 180,E1 -19572.243,E2 -19572.243} C_VEL
LIN {X 0,Y 250.622,Z 552.374,A -85,B 0,C 180,E1 -19575.488,E2 -19575.488} C_VEL
LIN {X 0,Y 250.77,Z 552.257,A -85,B 0,C 180,E1 -19577.731,E2 -19577.731} C_VEL
LIN {X 0,Y 251.357,Z 552.728,A -85,B 0,C 180,E1 -19579.978,E2 -19579.978} C_VEL
LIN {X 0,Y 252.27,Z 553.952,A -85,B 0,C 180,E1 -19582.201,E2 -19582.201} C_VEL
LIN {X 0,Y 253.634,Z 557.091,A -85,B 0,C 180,E1 -19585.215,E2 -19585.215} C_VEL
LIN {X 0,Y 255.12,Z 562.216,A -85,B 0,C 180,E1 -19588.439,E2 -19588.439} C_VEL
LIN {X 0,Y 255.847,Z 567.323,A -85,B 0,C 180,E1 -19590.927,E2 -19590.927} C_VEL
LIN {X 0,Y 256.064,Z 573.043,A -85,B 0,C 180,E1 -19593.416,E2 -19593.416} C_VEL
LIN {X 0,Y 255.792,Z 576.355,A -85,B 0,C 180,E1 -19594.794,E2 -19594.794} C_VEL
LIN {X 0,Y 254.6,Z 578.902,A -85,B 0,C 180,E1 -19595.54,E2 -19595.54} C_VEL
LIN {X 0,Y 250.338,Z 585.586,A -85,B 0,C 180,E1 -19597.728,E2 -19597.728} C_VEL
LIN {X 0,Y 246.499,Z 590.985,A -85,B 0,C 180,E1 -19599.993,E2 -19599.993} C_VEL
LIN {X 0,Y 243.153,Z 595.119,A -85,B 0,C 180,E1 -19602.333,E2 -19602.333} C_VEL
LIN {X 0,Y 240.287,Z 598.057,A -85,B 0,C 180,E1 -19604.738,E2 -19604.738} C_VEL
LIN {X 0,Y 238.547,Z 599.475,A -85,B 0,C 180,E1 -19606.471,E2 -19606.471} C_VEL
LIN {X 0,Y 235.856,Z 600.716,A -85,B 0,C 180,E1 -19609.701,E2 -19609.701} C_VEL
LIN {X 0,Y 234.958,Z 600.747,A -85,B 0,C 180,E1 -19611.399,E2 -19611.399} C_VEL
LIN {X 0,Y 234.317,Z 600.22,A -85,B 0,C 180,E1 -19613.11,E2 -19613.11} C_VEL
LIN {X 0,Y 233.785,Z 599.24,A -85,B 0,C 180,E1 -19614.826,E2 -19614.826} C_VEL
LIN {X 0,Y 233.377,Z 597.835,A -85,B 0,C 180,E1 -19616.547,E2 -19616.547} C_VEL
LIN {X 0,Y 232.981,Z 594.775,A -85,B 0,C 180,E1 -19619.136,E2 -19619.136} C_VEL
LIN {X 0,Y 232.974,Z 590.512,A -85,B 0,C 180,E1 -19621.729,E2 -19621.729} C_VEL
LIN {X 0,Y 233.126,Z 584.913,A -85,B 0,C 180,E1 -19624.322,E2 -19624.322} C_VEL
LIN {X 0,Y 233.487,Z 577.544,A -85,B 0,C 180,E1 -19626.915,E2 -19626.915} C_VEL
LIN {X 0,Y 233.883,Z 571.586,A -85,B 0,C 180,E1 -19628.641,E2 -19628.641} C_VEL
LIN {X 0,Y 234.34,Z 564.503,A -85,B 0,C 180,E1 -19630.367,E2 -19630.367} C_VEL
LIN {X 0,Y 235.058,Z 554.838,A -85,B 0,C 180,E1 -19632.3,E2 -19632.3} C_VEL
LIN {X 0,Y 235.877,Z 543.876,A -85,B 0,C 180,E1 -19634.01,E2 -19634.01} C_VEL
LIN {X 0,Y 235.589,Z 538.803,A -85,B 0,C 180,E1 -19634.689,E2 -19634.689} C_VEL
LIN {X 0,Y 234.149,Z 528.392,A -85,B 0,C 180,E1 -19635.817,E2 -19635.817} C_VEL
LIN {X 0,Y 233.213,Z 519.595,A -85,B 0,C 180,E1 -19636.574,E2 -19636.574} C_VEL
LIN {X 0,Y 233.17,Z 518.38,A -85,B 0,C 180,E1 -19638.109,E2 -19638.109} C_VEL
LIN {X 0,Y 234.732,Z 522.807,A -85,B 0,C 180,E1 -19641.849,E2 -19641.849} C_VEL
LIN {X 0,Y 236.236,Z 527.392,A -85,B 0,C 180,E1 -19645.555,E2 -19645.555} C_VEL
LIN {X 0,Y 236.425,Z 530.06,A -85,B 0,C 180,E1 -19647.526,E2 -19647.526} C_VEL
LIN {X 0,Y 236.239,Z 531.606,A -85,B 0,C 180,E1 -19648.606,E2 -19648.606} C_VEL
LIN {X 0,Y 239.623,Z 542.16,A -85,B 0,C 180,E1 -19649.908,E2 -19649.908} C_VEL
LIN {X 0,Y 241.882,Z 551.393,A -85,B 0,C 180,E1 -19651.169,E2 -19651.169} C_VEL
LIN {X 0,Y 243.238,Z 560.263,A -85,B 0,C 180,E1 -19652.506,E2 -19652.506} C_VEL
LIN {X 0,Y 243.926,Z 569.978,A -85,B 0,C 180,E1 -19654.183,E2 -19654.183} C_VEL
LIN {X 0,Y 243.583,Z 573.5,A -85,B 0,C 180,E1 -19654.841,E2 -19654.841} C_VEL
LIN {X 0,Y 241.649,Z 582.163,A -85,B 0,C 180,E1 -19656.54,E2 -19656.54} C_VEL
LIN {X 0,Y 239.725,Z 589.611,A -85,B 0,C 180,E1 -19658.391,E2 -19658.391} C_VEL
LIN {X 0,Y 237.893,Z 596.287,A -85,B 0,C 180,E1 -19660.537,E2 -19660.537} C_VEL
LIN {X 0,Y 236.291,Z 601.643,A -85,B 0,C 180,E1 -19662.724,E2 -19662.724} C_VEL
LIN {X 0,Y 234.96,Z 606.214,A -85,B 0,C 180,E1 -19665.172,E2 -19665.172} C_VEL
LIN {X 0,Y 233.997,Z 609.341,A -85,B 0,C 180,E1 -19667.484,E2 -19667.484} C_VEL
LIN {X 0,Y 233.016,Z 611.918,A -85,B 0,C 180,E1 -19670.699,E2 -19670.699} C_VEL
LIN {X 0,Y 232.621,Z 612.69,A -85,B 0,C 180,E1 -19672.824,E2 -19672.824} C_VEL
LIN {X 0,Y 232.426,Z 612.711,A -85,B 0,C 180,E1 -19674.933,E2 -19674.933} C_VEL
LIN {X 0,Y 232.441,Z 611.535,A -85,B 0,C 180,E1 -19677.844,E2 -19677.844} C_VEL
LIN {X 0,Y 232.75,Z 609.597,A -85,B 0,C 180,E1 -19680.117,E2 -19680.117} C_VEL
LIN {X 0,Y 233.154,Z 607.043,A -85,B 0,C 180,E1 -19682.145,E2 -19682.145} C_VEL
LIN {X 0,Y 233.678,Z 603.151,A -85,B 0,C 180,E1 -19684.458,E2 -19684.458} C_VEL
LIN {X 0,Y 234.556,Z 597.107,A -85,B 0,C 180,E1 -19687.074,E2 -19687.074} C_VEL
LIN {X 0,Y 235.405,Z 591.437,A -85,B 0,C 180,E1 -19689.006,E2 -19689.006} C_VEL
LIN {X 0,Y 236.23,Z 586.349,A -85,B 0,C 180,E1 -19690.445,E2 -19690.445} C_VEL
LIN {X 0,Y 237.236,Z 579.574,A -85,B 0,C 180,E1 -19692.044,E2 -19692.044} C_VEL
LIN {X 0,Y 238.379,Z 571.945,A -85,B 0,C 180,E1 -19693.514,E2 -19693.514} C_VEL
LIN {X 0,Y 239.055,Z 564.836,A -85,B 0,C 180,E1 -19694.656,E2 -19694.656} C_VEL
LIN {X 0,Y 238.172,Z 556.089,A -85,B 0,C 180,E1 -19695.909,E2 -19695.909} C_VEL
LIN {X 0,Y 236.738,Z 545.531,A -85,B 0,C 180,E1 -19697.134,E2 -19697.134} C_VEL
LIN {X 0,Y 234.634,Z 533.969,A -85,B 0,C 180,E1 -19698.115,E2 -19698.115} C_VEL
LIN {X 0,Y 234.15,Z 531.266,A -85,B 0,C 180,E1 -19698.31,E2 -19698.31} C_VEL
LIN {X 0,Y 234.679,Z 524.42,A -85,B 0,C 180,E1 -19703.119,E2 -19703.119} C_VEL
LIN {X 0,Y 235.064,Z 518.309,A -85,B 0,C 180,E1 -19707.429,E2 -19707.429} C_VEL
LIN {X 0,Y 235.37,Z 515.98,A -85,B 0,C 180,E1 -19709.144,E2 -19709.144} C_VEL
LIN {X 0,Y 235.598,Z 515.95,A -85,B 0,C 180,E1 -19711.709,E2 -19711.709} C_VEL
LIN {X 0,Y 235.407,Z 515.974,A -85,B 0,C 180,E1 -19716.858,E2 -19716.858} C_VEL
LIN {X 0,Y 235.255,Z 515.995,A -85,B 0,C 180,E1 -19720.325,E2 -19720.325} C_VEL
LIN {X 0,Y 235.115,Z 516.009,A -85,B 0,C 180,E1 -19725.605,E2 -19725.605} C_VEL
LIN {X 0,Y 235.009,Z 516.02,A -85,B 0,C 180,E1 -19729.205,E2 -19729.205} C_VEL
LIN {X 0,Y 234.961,Z 516.026,A -85,B 0,C 180,E1 -19732.882,E2 -19732.882} C_VEL
LIN {X 0,Y 234.971,Z 516.027,A -85,B 0,C 180,E1 -19736.656,E2 -19736.656} C_VEL
LIN {X 0,Y 234.932,Z 516.033,A -85,B 0,C 180,E1 -19740.567,E2 -19740.567} C_VEL
LIN {X 0,Y 234.96,Z 516.027,A -85,B 0,C 180,E1 -19744.632,E2 -19744.632} C_VEL
LIN {X 0,Y 234.94,Z 516.03,A -85,B 0,C 180,E1 -19748.944,E2 -19748.944} C_VEL
LIN {X 0,Y 234.959,Z 516.024,A -85,B 0,C 180,E1 -19753.468,E2 -19753.468} C_VEL
LIN {X 0,Y 234.964,Z 516.028,A -85,B 0,C 180,E1 -19756.532,E2 -19756.532} C_VEL
LIN {X 0,Y 234.953,Z 516.026,A -85,B 0,C 180,E1 -19761.085,E2 -19761.085} C_VEL
LIN {X 0,Y 234.959,Z 516.026,A -85,B 0,C 180,E1 -19765.367,E2 -19765.367} C_VEL
LIN {X 0,Y 234.921,Z 516.034,A -85,B 0,C 180,E1 -19769.431,E2 -19769.431} C_VEL
LIN {X 0,Y 234.991,Z 516.024,A -85,B 0,C 180,E1 -19773.793,E2 -19773.793} C_VEL
LIN {X 0,Y 235.009,Z 516.021,A -85,B 0,C 180,E1 -19778.969,E2 -19778.969} C_VEL
LIN {X 0,Y 235.094,Z 516.01,A -85,B 0,C 180,E1 -19783.059,E2 -19783.059} C_VEL
LIN {X 0,Y 235.145,Z 516.006,A -85,B 0,C 180,E1 -19787.923,E2 -19787.923} C_VEL
LIN {X 0,Y 235.388,Z 515.975,A -85,B 0,C 180,E1 -19791.414,E2 -19791.414} C_VEL
LIN {X 0,Y 235.404,Z 515.973,A -85,B 0,C 180,E1 -19793.141,E2 -19793.141} C_VEL
LIN {X 0,Y 235.595,Z 515.944,A -85,B 0,C 180,E1 -19798.29,E2 -19798.29} C_VEL
LIN {X 0,Y 235.595,Z 515.95,A -85,B 0,C 180,E1 -19801.709,E2 -19801.709} C_VEL
LIN {X 0,Y 235.404,Z 515.971,A -85,B 0,C 180,E1 -19806.859,E2 -19806.859} C_VEL
LIN {X 0,Y 235.251,Z 515.992,A -85,B 0,C 180,E1 -19810.326,E2 -19810.326} C_VEL
LIN {X 0,Y 235.111,Z 516.013,A -85,B 0,C 180,E1 -19815.606,E2 -19815.606} C_VEL
LIN {X 0,Y 235.007,Z 516.024,A -85,B 0,C 180,E1 -19819.206,E2 -19819.206} C_VEL
LIN {X 0,Y 234.959,Z 516.03,A -85,B 0,C 180,E1 -19822.883,E2 -19822.883} C_VEL
LIN {X 0,Y 234.967,Z 516.028,A -85,B 0,C 180,E1 -19826.658,E2 -19826.658} C_VEL
LIN {X 0,Y 234.929,Z 516.033,A -85,B 0,C 180,E1 -19830.568,E2 -19830.568} C_VEL
LIN {X 0,Y 234.958,Z 516.028,A -85,B 0,C 180,E1 -19834.633,E2 -19834.633} C_VEL
LIN {X 0,Y 234.939,Z 516.031,A -85,B 0,C 180,E1 -19838.945,E2 -19838.945} C_VEL
LIN {X 0,Y 234.921,Z 516.038,A -85,B 0,C 180,E1 -19843.478,E2 -19843.478} C_VEL
LIN {X 0,Y 234.955,Z 516.029,A -85,B 0,C 180,E1 -19846.531,E2 -19846.531} C_VEL
LIN {X 0,Y 235.188,Z 516.002,A -85,B 0,C 180,E1 -19851.954,E2 -19851.954} C_VEL
LIN {X 0,Y 235.048,Z 516.38,A -85,B 0,C 180,E1 -19852.91,E2 -19852.91} C_VEL
LIN {X 0,Y 234.451,Z 517.283,A -85,B 0,C 180,E1 -19853.843,E2 -19853.843} C_VEL
LIN {X 0,Y 232.439,Z 519.627,A -85,B 0,C 180,E1 -19855.655,E2 -19855.655} C_VEL
LIN {X 0,Y 229.301,Z 523.166,A -85,B 0,C 180,E1 -19858.412,E2 -19858.412} C_VEL
LIN {X 0,Y 228.777,Z 524.324,A -85,B 0,C 180,E1 -19859.365,E2 -19859.365} C_VEL
LIN {X 0,Y 227.522,Z 530.445,A -85,B 0,C 180,E1 -19864.378,E2 -19864.378} C_VEL
LIN {X 0,Y 227.197,Z 532.551,A -85,B 0,C 180,E1 -19866.047,E2 -19866.047} C_VEL
LIN {X 0,Y 227.229,Z 536.7,A -85,B 0,C 180,E1 -19867.145,E2 -19867.145} C_VEL
LIN {X 0,Y 229.093,Z 550.612,A -85,B 0,C 180,E1 -19868.005,E2 -19868.005} C_VEL
LIN {X 0,Y 229.909,Z 560.013,A -85,B 0,C 180,E1 -19868.834,E2 -19868.834} C_VEL
LIN {X 0,Y 230.442,Z 569.655,A -85,B 0,C 180,E1 -19869.935,E2 -19869.935} C_VEL
LIN {X 0,Y 230.682,Z 578.131,A -85,B 0,C 180,E1 -19871.146,E2 -19871.146} C_VEL
LIN {X 0,Y 230.418,Z 587.077,A -85,B 0,C 180,E1 -19872.7,E2 -19872.7} C_VEL
LIN {X 0,Y 229.128,Z 595.217,A -85,B 0,C 180,E1 -19874.433,E2 -19874.433} C_VEL
LIN {X 0,Y 228.071,Z 601.784,A -85,B 0,C 180,E1 -19876.184,E2 -19876.184} C_VEL
LIN {X 0,Y 227.084,Z 608.407,A -85,B 0,C 180,E1 -19878.396,E2 -19878.396} C_VEL
LIN {X 0,Y 226.514,Z 612.737,A -85,B 0,C 180,E1 -19880.175,E2 -19880.175} C_VEL
LIN {X 0,Y 225.931,Z 617.823,A -85,B 0,C 180,E1 -19882.853,E2 -19882.853} C_VEL
LIN {X 0,Y 225.717,Z 620.964,A -85,B 0,C 180,E1 -19885.109,E2 -19885.109} C_VEL
LIN {X 0,Y 225.72,Z 623.768,A -85,B 0,C 180,E1 -19888.217,E2 -19888.217} C_VEL
LIN {X 0,Y 225.791,Z 624.676,A -85,B 0,C 180,E1 -19890.001,E2 -19890.001} C_VEL
LIN {X 0,Y 225.699,Z 624.983,A -85,B 0,C 180,E1 -19891.785,E2 -19891.785} C_VEL
LIN {X 0,Y 225.716,Z 624.378,A -85,B 0,C 180,E1 -19894.886,E2 -19894.886} C_VEL
LIN {X 0,Y 226.01,Z 622.964,A -85,B 0,C 180,E1 -19897.146,E2 -19897.146} C_VEL
LIN {X 0,Y 226.722,Z 620.157,A -85,B 0,C 180,E1 -19899.817,E2 -19899.817} C_VEL
LIN {X 0,Y 227.246,Z 618.67,A -85,B 0,C 180,E1 -19901.146,E2 -19901.146} C_VEL
LIN {X 0,Y 227.929,Z 618.223,A -85,B 0,C 180,E1 -19902.466,E2 -19902.466} C_VEL
LIN {X 0,Y 229.062,Z 617.088,A -85,B 0,C 180,E1 -19904.21,E2 -19904.21} C_VEL
LIN {X 0,Y 232.188,Z 613.626,A -85,B 0,C 180,E1 -19907.62,E2 -19907.62} C_VEL
LIN {X 0,Y 235.221,Z 609.763,A -85,B 0,C 180,E1 -19910.097,E2 -19910.097} C_VEL
LIN {X 0,Y 238.744,Z 604.788,A -85,B 0,C 180,E1 -19912.501,E2 -19912.501} C_VEL
LIN {X 0,Y 242.142,Z 599.715,A -85,B 0,C 180,E1 -19914.432,E2 -19914.432} C_VEL
LIN {X 0,Y 244.533,Z 594.823,A -85,B 0,C 180,E1 -19916.121,E2 -19916.121} C_VEL
LIN {X 0,Y 246.277,Z 589.221,A -85,B 0,C 180,E1 -19918.09,E2 -19918.09} C_VEL
LIN {X 0,Y 247.624,Z 581.739,A -85,B 0,C 180,E1 -19920.723,E2 -19920.723} C_VEL
LIN {X 0,Y 248.216,Z 575.653,A -85,B 0,C 180,E1 -19922.971,E2 -19922.971} C_VEL
LIN {X 0,Y 248.465,Z 570.91,A -85,B 0,C 180,E1 -19924.887,E2 -19924.887} C_VEL
LIN {X 0,Y 248.384,Z 567.552,A -85,B 0,C 180,E1 -19926.456,E2 -19926.456} C_VEL
LIN {X 0,Y 248.033,Z 563.868,A -85,B 0,C 180,E1 -19928.563,E2 -19928.563} C_VEL
LIN {X 0,Y 247.339,Z 561.411,A -85,B 0,C 180,E1 -19930.81,E2 -19930.81} C_VEL
LIN {X 0,Y 246.934,Z 559.58,A -85,B 0,C 180,E1 -19933.085,E2 -19933.085} C_VEL
LIN {X 0,Y 246.873,Z 558.447,A -85,B 0,C 180,E1 -19935.375,E2 -19935.375} C_VEL
LIN {X 0,Y 247.002,Z 558.274,A -85,B 0,C 180,E1 -19937.714,E2 -19937.714} C_VEL
LIN {X 0,Y 247.507,Z 558.717,A -85,B 0,C 180,E1 -19940.057,E2 -19940.057} C_VEL
LIN {X 0,Y 248.259,Z 560.037,A -85,B 0,C 180,E1 -19942.436,E2 -19942.436} C_VEL
LIN {X 0,Y 249.193,Z 562.43,A -85,B 0,C 180,E1 -19944.875,E2 -19944.875} C_VEL
LIN {X 0,Y 250.026,Z 566.433,A -85,B 0,C 180,E1 -19947.719,E2 -19947.719} C_VEL
LIN {X 0,Y 250.439,Z 571.432,A -85,B 0,C 180,E1 -19950.454,E2 -19950.454} C_VEL
LIN {X 0,Y 250.351,Z 575.8,A -85,B 0,C 180,E1 -19952.569,E2 -19952.569} C_VEL
LIN {X 0,Y 249.949,Z 579.239,A -85,B 0,C 180,E1 -19954.129,E2 -19954.129} C_VEL
LIN {X 0,Y 245.498,Z 585.95,A -85,B 0,C 180,E1 -19956.373,E2 -19956.373} C_VEL
LIN {X 0,Y 241.347,Z 591.303,A -85,B 0,C 180,E1 -19958.654,E2 -19958.654} C_VEL
LIN {X 0,Y 237.686,Z 595.438,A -85,B 0,C 180,E1 -19961.019,E2 -19961.019} C_VEL
LIN {X 0,Y 235.465,Z 597.515,A -85,B 0,C 180,E1 -19962.634,E2 -19962.634} C_VEL
LIN {X 0,Y 233.525,Z 599.129,A -85,B 0,C 180,E1 -19964.285,E2 -19964.285} C_VEL
LIN {X 0,Y 231.611,Z 600.411,A -85,B 0,C 180,E1 -19966.173,E2 -19966.173} C_VEL
LIN {X 0,Y 230.323,Z 601.021,A -85,B 0,C 180,E1 -19967.667,E2 -19967.667} C_VEL
LIN {X 0,Y 228.905,Z 601.234,A -85,B 0,C 180,E1 -19969.385,E2 -19969.385} C_VEL
LIN {X 0,Y 227.949,Z 601.023,A -85,B 0,C 180,E1 -19971.132,E2 -19971.132} C_VEL
LIN {X 0,Y 227.266,Z 600.413,A -85,B 0,C 180,E1 -19972.895,E2 -19972.895} C_VEL
LIN {X 0,Y 226.725,Z 599.265,A -85,B 0,C 180,E1 -19974.664,E2 -19974.664} C_VEL
LIN {X 0,Y 226.134,Z 596.716,A -85,B 0,C 180,E1 -19977.328,E2 -19977.328} C_VEL
LIN {X 0,Y 225.879,Z 592.969,A -85,B 0,C 180,E1 -19980,E2 -19980} C_VEL
LIN {X 0,Y 225.979,Z 587.956,A -85,B 0,C 180,E1 -19982.674,E2 -19982.674} C_VEL
LIN {X 0,Y 226.111,Z 582.638,A -85,B 0,C 180,E1 -19984.904,E2 -19984.904} C_VEL
LIN {X 0,Y 226.48,Z 576.123,A -85,B 0,C 180,E1 -19987.13,E2 -19987.13} C_VEL
LIN {X 0,Y 226.983,Z 568.154,A -85,B 0,C 180,E1 -19989.355,E2 -19989.355} C_VEL
LIN {X 0,Y 227.631,Z 559.191,A -85,B 0,C 180,E1 -19991.352,E2 -19991.352} C_VEL
LIN {X 0,Y 228.3,Z 550.815,A -85,B 0,C 180,E1 -19992.896,E2 -19992.896} C_VEL
LIN {X 0,Y 228.881,Z 542.146,A -85,B 0,C 180,E1 -19994.22,E2 -19994.22} C_VEL
LIN {X 0,Y 227.306,Z 530.972,A -85,B 0,C 180,E1 -19995.581,E2 -19995.581} C_VEL
LIN {X 0,Y 226.142,Z 519.924,A -85,B 0,C 180,E1 -19996.591,E2 -19996.591} C_VEL
LIN {X 0,Y 226.11,Z 519.467,A -85,B 0,C 180,E1 -19997.175,E2 -19997.175} C_VEL
LIN {X 0,Y 227.861,Z 524.633,A -85,B 0,C 180,E1 -20001.723,E2 -20001.723} C_VEL
LIN {X 0,Y 229.341,Z 529.049,A -85,B 0,C 180,E1 -20005.406,E2 -20005.406} C_VEL
LIN {X 0,Y 229.526,Z 531.746,A -85,B 0,C 180,E1 -20007.454,E2 -20007.454} C_VEL
LIN {X 0,Y 232.985,Z 542.359,A -85,B 0,C 180,E1 -20008.858,E2 -20008.858} C_VEL
